C07268=1101.873,173.117,-65.868,177.861,15.228,151.662
C07269=1101.878,173.366,-65.890,177.865,15.228,151.661
C07270=1101.885,173.615,-65.912,177.869,15.227,151.660
C07271=1101.890,173.864,-65.934,177.872,15.226,151.659
C07272=1101.895,174.113,-65.957,177.876,15.226,151.658
C07273=1101.902,174.362,-65.979,177.880,15.225,151.657
C07274=1101.907,174.611,-66.002,177.883,15.224,151.656
C07275=1101.913,174.860,-66.024,177.887,15.224,151.655
C07276=1101.918,175.108,-66.046,177.890,15.223,151.654
C07277=1101.924,175.358,-66.068,177.895,15.222,151.653
C07278=1101.930,175.606,-66.091,177.898,15.222,151.652
C07279=1101.936,175.879,-66.115,177.902,15.222,151.652
C07280=1101.942,176.151,-66.140,177.906,15.221,151.650
C07281=1101.948,176.424,-66.164,177.910,15.220,151.649
C07282=1101.955,176.697,-66.188,177.914,15.219,151.648
C07283=1101.960,176.946,-66.211,177.918,15.219,151.647
C07284=1101.966,177.194,-66.234,177.922,15.218,151.647
C07285=1101.972,177.443,-66.256,177.925,15.217,151.646
C07286=1101.977,177.692,-66.279,177.929,15.217,151.645
C07287=1101.983,177.941,-66.302,177.932,15.216,151.644
C07288=1101.989,178.190,-66.323,177.936,15.215,151.643
C07289=1101.995,178.439,-66.346,177.940,15.215,151.642
C07290=1102.000,178.688,-66.369,177.943,15.214,151.641
C07291=1102.006,178.937,-66.391,177.947,15.213,151.640
C07292=1102.011,179.186,-66.414,177.952,15.213,151.639
C07293=1102.018,179.435,-66.436,177.955,15.212,151.638
C07294=1102.023,179.684,-66.458,177.959,15.211,151.637
C07295=1102.029,179.933,-66.481,177.963,15.211,151.636
C07296=1102.035,180.182,-66.504,177.966,15.210,151.635
C07297=1102.041,180.430,-66.527,177.970,15.209,151.634
C07298=1102.047,180.679,-66.550,177.973,15.208,151.633
C07299=1102.052,180.928,-66.572,177.977,15.208,151.632
C07300=1102.057,181.177,-66.594,177.981,15.207,151.631
C07301=1102.063,181.426,-66.617,177.984,15.206,151.630
C07302=1102.069,181.675,-66.640,177.989,15.205,151.629
C07303=1102.075,181.923,-66.663,177.992,15.205,151.629
C07304=1102.081,182.173,-66.685,177.996,15.204,151.628
C07305=1102.087,182.422,-66.708,178.000,15.203,151.627
C07306=1102.092,182.671,-66.731,178.004,15.203,151.626
C07307=1102.098,182.920,-66.754,178.007,15.202,151.625
C07308=1102.104,183.169,-66.777,178.011,15.201,151.624
C07309=1102.110,183.417,-66.799,178.014,15.200,151.623
C07310=1102.116,183.666,-66.822,178.018,15.200,151.622
C07311=1102.122,183.915,-66.845,178.022,15.199,151.621
C07312=1102.127,184.164,-66.868,178.026,15.198,151.620
C07313=1102.133,184.413,-66.891,178.030,15.197,151.619
C07314=1102.139,184.662,-66.914,178.034,15.197,151.618
C07315=1102.144,184.911,-66.936,178.037,15.196,151.617
C07316=1102.150,185.160,-66.959,178.041,15.195,151.616
C07317=1102.156,185.409,-66.982,178.045,15.195,151.615
C07318=1102.161,185.658,-67.005,178.048,15.194,151.614
C07319=1102.167,185.907,-67.028,178.052,15.193,151.613
C07320=1102.172,186.155,-67.050,178.056,15.193,151.612
C07321=1102.178,186.404,-67.073,178.059,15.192,151.611
C07322=1102.183,186.653,-67.097,178.064,15.191,151.610
C07323=1102.189,186.902,-67.120,178.068,15.191,151.609
C07324=1102.195,187.150,-67.143,178.071,15.190,151.608
C07325=1102.201,187.399,-67.166,178.075,15.189,151.607
C07326=1102.206,187.648,-67.189,178.079,15.189,151.606
C07327=1102.211,187.897,-67.213,178.082,15.188,151.605
C07328=1102.217,188.146,-67.236,178.086,15.187,151.604
C07329=1102.223,188.395,-67.259,178.090,15.187,151.603
C07330=1102.228,188.644,-67.282,178.093,15.186,151.603
C07331=1102.234,188.893,-67.305,178.098,15.185,151.601
C07332=1102.239,189.142,-67.328,178.101,15.185,151.601
C07333=1102.245,189.391,-67.351,178.105,15.183,151.600
C07334=1102.251,189.639,-67.375,178.109,15.183,151.599
C07335=1102.257,189.888,-67.398,178.113,15.182,151.598
C07336=1102.262,190.137,-67.421,178.116,15.182,151.597
C07337=1102.267,190.386,-67.444,178.120,15.181,151.596
C07338=1102.273,190.635,-67.467,178.124,15.181,151.595
C07339=1102.279,190.883,-67.491,178.128,15.179,151.594
C07340=1102.284,191.133,-67.514,178.132,15.179,151.593
C07341=1102.290,191.381,-67.537,178.136,15.178,151.592
C07342=1102.296,191.630,-67.560,178.139,15.177,151.591
C07343=1102.302,191.902,-67.587,178.143,15.176,151.590
C07344=1102.308,192.174,-67.611,178.147,15.176,151.589
C07345=1102.314,192.447,-67.637,178.152,15.175,151.588
C07346=1102.321,192.719,-67.663,178.156,15.174,151.586
C07347=1102.326,192.968,-67.686,178.160,15.173,151.585
C07348=1102.332,193.216,-67.710,178.163,15.173,151.585
C07349=1102.337,193.465,-67.733,178.167,15.172,151.583
C07350=1102.342,193.714,-67.756,178.172,15.171,151.582
C07351=1102.348,193.962,-67.780,178.175,15.170,151.582
C07352=1102.354,194.211,-67.803,178.179,15.170,151.580
C07353=1102.360,194.461,-67.827,178.183,15.169,151.579
C07354=1102.366,194.710,-67.850,178.186,15.168,151.579
C07355=1102.371,194.958,-67.873,178.190,15.167,151.578
C07356=1102.377,195.207,-67.898,178.195,15.167,151.576
C07357=1102.382,195.456,-67.921,178.198,15.165,151.575
C07358=1102.388,195.704,-67.944,178.202,15.165,151.575
C07359=1102.393,195.953,-67.968,178.206,15.164,151.573
C07360=1102.400,196.203,-67.991,178.210,15.164,151.572
C07361=1102.406,196.451,-68.015,178.213,15.163,151.572
C07362=1102.411,196.700,-68.038,178.218,15.162,151.570
C07363=1102.417,196.949,-68.062,178.222,15.161,151.569
C07364=1102.422,197.198,-68.086,178.225,15.160,151.568
C07365=1102.428,197.446,-68.109,178.229,15.159,151.567
C07366=1102.435,197.695,-68.133,178.233,15.159,151.566
C07367=1102.440,197.944,-68.157,178.237,15.158,151.565
C07368=1102.446,198.193,-68.180,178.241,15.157,151.564
C07369=1102.451,198.442,-68.204,178.245,15.156,151.563
C07370=1102.457,198.690,-68.228,178.248,15.155,151.562
C07371=1102.462,198.940,-68.252,178.252,15.155,151.561
C07372=1102.468,199.188,-68.275,178.257,15.154,151.560
C07373=1102.474,199.437,-68.299,178.260,15.153,151.559
C07374=1102.479,199.686,-68.322,178.264,15.152,151.558
C07375=1102.485,199.934,-68.346,178.268,15.151,151.557
C07376=1102.491,200.183,-68.371,178.272,15.150,151.556
C07377=1102.497,200.432,-68.394,178.276,15.150,151.555
C07378=1102.502,200.681,-68.418,178.280,15.149,151.554
C07379=1102.509,200.930,-68.442,178.283,15.148,151.553
C07380=1102.514,201.179,-68.465,178.288,15.147,151.552
C07381=1102.520,201.427,-68.489,178.292,15.146,151.551
C07382=1102.525,201.676,-68.513,178.295,15.145,151.550
C07383=1102.532,201.925,-68.537,178.299,15.144,151.549
C07384=1102.537,202.174,-68.561,178.304,15.144,151.548
C07385=1102.543,202.422,-68.585,178.308,15.143,151.547
C07386=1102.549,202.672,-68.609,178.311,15.142,151.546
C07387=1102.555,202.920,-68.633,178.315,15.141,151.545
C07388=1102.560,203.169,-68.657,178.319,15.141,151.544
C07389=1102.565,203.418,-68.681,178.323,15.140,151.543
C07390=1102.572,203.667,-68.705,178.327,15.139,151.542
C07391=1102.577,203.915,-68.729,178.331,15.138,151.541
C07392=1102.582,204.164,-68.753,178.334,15.137,151.540
C07393=1102.588,204.412,-68.777,178.339,15.136,151.539
C07394=1102.594,204.661,-68.801,178.343,15.136,151.538
C07395=1102.600,204.910,-68.826,178.346,15.134,151.536
C07396=1102.605,205.159,-68.849,178.350,15.134,151.535
C07397=1102.611,205.408,-68.873,178.354,15.133,151.535
C07398=1102.617,205.657,-68.898,178.359,15.133,151.533
C07399=1102.622,205.905,-68.922,178.362,15.131,151.532
C07400=1102.628,206.154,-68.945,178.366,15.131,151.531
C07401=1102.634,206.403,-68.970,178.370,15.130,151.530
C07402=1102.639,206.652,-68.994,178.374,15.129,151.529
C07403=1102.644,206.900,-69.019,178.378,15.128,151.528
C07404=1102.651,207.149,-69.043,178.382,15.127,151.527
C07405=1102.656,207.398,-69.067,178.386,15.127,151.526
C07406=1102.662,207.647,-69.092,178.390,15.125,151.525
C07407=1102.685,208.648,-69.188,178.422,15.131,151.519
C07408=1102.693,209.016,-69.225,178.428,15.131,151.518
C07409=1102.702,209.384,-69.261,178.434,15.131,151.517
C07410=1102.710,209.752,-69.297,178.439,15.131,151.516
C07411=1102.718,210.119,-69.333,178.445,15.131,151.515
C07412=1102.724,210.369,-69.358,178.448,15.132,151.514
C07413=1102.730,210.617,-69.383,178.451,15.131,151.513
C07414=1102.736,210.866,-69.408,178.455,15.131,151.512
C07415=1102.741,211.114,-69.432,178.459,15.131,151.511
C07416=1102.746,211.363,-69.456,178.462,15.131,151.511
C07417=1102.753,211.612,-69.481,178.466,15.131,151.510
C07418=1102.758,211.860,-69.506,178.470,15.131,151.509
C07419=1102.764,212.110,-69.530,178.474,15.131,151.508
C07420=1102.769,212.358,-69.555,178.477,15.131,151.507
C07421=1102.775,212.607,-69.580,178.481,15.131,151.507
C07422=1102.781,212.855,-69.604,178.485,15.132,151.506
C07423=1102.786,213.105,-69.629,178.489,15.131,151.505
C07424=1102.792,213.353,-69.654,178.493,15.132,151.504
C07425=1102.798,213.602,-69.678,178.497,15.131,151.503
C07426=1102.803,213.851,-69.703,178.500,15.132,151.503
C07427=1102.809,214.099,-69.728,178.504,15.131,151.502
C07428=1102.815,214.348,-69.752,178.508,15.132,151.501
C07429=1102.820,214.596,-69.778,178.511,15.132,151.500
C07430=1102.825,214.845,-69.802,178.515,15.132,151.499
C07431=1102.831,215.094,-69.827,178.519,15.132,151.499
C07432=1102.837,215.343,-69.852,178.522,15.132,151.498
C07433=1102.842,215.591,-69.876,178.526,15.132,151.497
C07434=1102.849,215.840,-69.902,178.530,15.132,151.496
C07435=1102.853,216.089,-69.927,178.533,15.132,151.496
C07436=1102.859,216.337,-69.952,178.537,15.132,151.495
C07437=1102.865,216.586,-69.976,178.541,15.132,151.494
C07438=1102.871,216.835,-70.001,178.544,15.132,151.493
C07439=1102.877,217.084,-70.026,178.548,15.132,151.492
C07440=1102.882,217.332,-70.051,178.552,15.132,151.492
C07441=1102.887,217.582,-70.076,178.556,15.132,151.491
C07442=1102.893,217.830,-70.101,178.559,15.132,151.490
C07443=1102.899,218.079,-70.126,178.563,15.132,151.489
C07444=1102.905,218.327,-70.151,178.567,15.132,151.488
C07445=1102.910,218.576,-70.177,178.571,15.132,151.488
C07446=1102.916,218.825,-70.201,178.574,15.132,151.487
C07447=1102.922,219.073,-70.226,178.578,15.133,151.486
C07448=1102.927,219.322,-70.251,178.581,15.132,151.485
C07449=1102.932,219.571,-70.277,178.585,15.133,151.485
C07450=1102.938,219.819,-70.302,178.589,15.132,151.484
C07451=1102.944,220.069,-70.326,178.592,15.133,151.483
C07452=1102.950,220.317,-70.351,178.596,15.132,151.482
C07453=1102.955,220.566,-70.377,178.600,15.133,151.481
C07454=1102.961,220.814,-70.402,178.604,15.132,151.480
C07455=1102.967,221.063,-70.427,178.607,15.133,151.480
C07456=1102.973,221.311,-70.452,178.612,15.133,151.479
C07457=1102.978,221.560,-70.478,178.615,15.133,151.478
C07458=1102.984,221.809,-70.503,178.619,15.133,151.477
C07459=1102.990,222.058,-70.528,178.623,15.133,151.477
C07460=1102.998,222.429,-70.566,178.628,15.133,151.475
C07461=1103.007,222.800,-70.603,178.634,15.134,151.474
C07462=1103.015,223.171,-70.641,178.639,15.133,151.473
C07463=1103.023,223.543,-70.680,178.645,15.134,151.472
C07464=1103.029,223.792,-70.704,178.649,15.134,151.471
C07465=1103.034,224.041,-70.730,178.652,15.134,151.470
C07466=1103.040,224.289,-70.756,178.656,15.134,151.470
C07467=1103.046,224.537,-70.781,178.660,15.134,151.469
C07468=1103.051,224.786,-70.806,178.663,15.134,151.468
C07469=1103.058,225.035,-70.832,178.667,15.134,151.467
C07470=1103.062,225.283,-70.857,178.671,15.135,151.466
C07471=1103.069,225.532,-70.883,178.675,15.135,151.466
C07472=1103.074,225.781,-70.909,178.679,15.135,151.465
C07473=1103.080,226.029,-70.934,178.682,15.135,151.464
C07474=1103.085,226.278,-70.960,178.686,15.135,151.463
C07475=1103.091,226.527,-70.985,178.690,15.135,151.463
C07476=1103.097,226.776,-71.011,178.693,15.136,151.462
C07477=1103.102,227.024,-71.036,178.697,15.135,151.461
C07478=1103.108,227.272,-71.062,178.701,15.136,151.460
C07479=1103.113,227.521,-71.088,178.704,15.136,151.459
C07480=1103.120,227.770,-71.113,178.708,15.136,151.459
C07481=1103.125,228.018,-71.139,178.712,15.137,151.458
C07482=1103.131,228.267,-71.164,178.716,15.137,151.457
C07483=1103.136,228.516,-71.190,178.720,15.137,151.456
C07484=1103.142,228.765,-71.215,178.724,15.137,151.455
C07485=1103.148,229.014,-71.241,178.727,15.137,151.455
C07486=1103.153,229.262,-71.267,178.731,15.137,151.454
C07487=1103.159,229.511,-71.292,178.735,15.137,151.453
C07488=1103.165,229.759,-71.319,178.738,15.137,151.452
C07489=1103.171,230.008,-71.344,178.742,15.137,151.452
C07490=1103.176,230.257,-71.370,178.746,15.137,151.451
C07491=1103.181,230.505,-71.396,178.749,15.138,151.450
C07492=1103.187,230.754,-71.421,178.754,15.138,151.449
C07493=1103.193,231.002,-71.448,178.757,15.138,151.449
C07494=1103.199,231.251,-71.473,178.761,15.138,151.448
C07495=1103.205,231.500,-71.499,178.765,15.138,151.447
C07496=1103.210,231.748,-71.524,178.768,15.139,151.446
C07497=1103.215,231.997,-71.550,178.772,15.139,151.446
C07498=1103.221,232.245,-71.577,178.776,15.139,151.445
C07499=1103.227,232.494,-71.602,178.779,15.139,151.444
C07500=1103.233,232.743,-71.628,178.783,15.140,151.443
C07501=1103.238,232.991,-71.655,178.787,15.140,151.442
C07502=1103.243,233.240,-71.680,178.791,15.140,151.442
C07503=1103.249,233.489,-71.706,178.794,15.140,151.441
C07504=1103.255,233.737,-71.732,178.798,15.140,151.440
C07505=1103.261,233.986,-71.758,178.802,15.140,151.439
C07506=1103.266,234.235,-71.784,178.805,15.141,151.439
C07507=1103.272,234.483,-71.811,178.809,15.140,151.438
C07508=1103.277,234.732,-71.837,178.813,15.141,151.437
C07509=1103.284,234.981,-71.862,178.817,15.142,151.436
C07510=1103.289,235.228,-71.888,178.821,15.142,151.436
C07511=1103.294,235.477,-71.914,178.824,15.142,151.435
C07512=1103.303,235.841,-71.953,178.830,15.142,151.434
C07513=1103.311,236.203,-71.992,178.835,15.142,151.433
C07514=1103.319,236.566,-72.030,178.841,15.143,151.432
C07515=1103.327,236.929,-72.068,178.846,15.143,151.430
C07516=1103.333,237.178,-72.094,178.850,15.144,151.430
C07517=1103.339,237.426,-72.120,178.854,15.144,151.429
C07518=1103.344,237.675,-72.146,178.858,15.144,151.428
C07519=1103.350,237.923,-72.173,178.861,15.144,151.427
C07520=1103.356,238.172,-72.199,178.865,15.144,151.427
C07521=1103.361,238.421,-72.225,178.868,15.145,151.426
C07522=1103.367,238.669,-72.252,178.873,15.145,151.425
C07523=1103.372,238.918,-72.278,178.876,15.145,151.424
C07524=1103.378,239.166,-72.305,178.880,15.146,151.424
C07525=1103.384,239.415,-72.331,178.884,15.145,151.423
C07526=1103.389,239.664,-72.357,178.887,15.146,151.422
C07527=1103.395,239.912,-72.384,178.891,15.146,151.421
C07528=1103.401,240.160,-72.410,178.895,15.147,151.421
C07529=1103.406,240.409,-72.436,178.899,15.147,151.420
C07530=1103.412,240.658,-72.463,178.903,15.147,151.419
C07531=1103.418,240.906,-72.490,178.906,15.147,151.418
C07532=1103.423,241.155,-72.516,178.910,15.147,151.418
C07533=1103.429,241.403,-72.542,178.914,15.147,151.417
C07534=1103.435,241.652,-72.569,178.918,15.148,151.416
C07535=1103.441,241.900,-72.596,178.921,15.149,151.415
C07536=1103.446,242.148,-72.622,178.925,15.149,151.415
C07537=1103.452,242.397,-72.648,178.929,15.149,151.414
C07538=1103.458,242.646,-72.675,178.932,15.149,151.413
C07539=1103.463,242.894,-72.701,178.936,15.149,151.412
C07540=1103.469,243.143,-72.728,178.940,15.150,151.412
C07541=1103.475,243.391,-72.755,178.944,15.150,151.411
C07542=1103.480,243.640,-72.781,178.947,15.150,151.410
C07543=1103.486,243.889,-72.808,178.951,15.151,151.409
C07544=1103.491,244.137,-72.835,178.955,15.151,151.409
C07545=1103.497,244.385,-72.861,178.959,15.152,151.408
C07546=1103.503,244.634,-72.888,178.963,15.152,151.407
C07547=1103.508,244.883,-72.915,178.966,15.152,151.406
C07548=1103.514,245.131,-72.942,178.970,15.152,151.406
C07549=1103.520,245.380,-72.969,178.973,15.153,151.405
C07550=1103.526,245.628,-72.995,178.978,15.154,151.404
C07551=1103.532,245.876,-73.022,178.981,15.153,151.403
C07552=1103.537,246.125,-73.049,178.985,15.154,151.403
C07553=1103.542,246.373,-73.076,178.989,15.154,151.402
C07554=1103.548,246.622,-73.103,178.992,15.154,151.401
C07555=1103.553,246.871,-73.130,178.996,15.155,151.401
C07556=1103.559,247.119,-73.156,179.000,15.155,151.400
C07557=1103.565,247.367,-73.183,179.004,15.155,151.399
C07558=1103.571,247.616,-73.210,179.007,15.156,151.398
C07559=1103.576,247.865,-73.237,179.012,15.157,151.398
C07560=1103.582,248.113,-73.264,179.015,15.157,151.397
C07561=1103.587,248.362,-73.291,179.019,15.157,151.396
C07562=1103.593,248.610,-73.318,179.022,15.157,151.396
C07563=1103.599,248.859,-73.345,179.026,15.158,151.395
C07564=1103.607,249.215,-73.384,179.031,15.158,151.394
C07565=1103.614,249.572,-73.422,179.037,15.159,151.393
C07566=1103.623,249.928,-73.461,179.042,15.160,151.392
C07567=1103.630,250.283,-73.500,179.047,15.161,151.391
C07568=1103.636,250.532,-73.527,179.051,15.161,151.390
C07569=1103.641,250.780,-73.554,179.055,15.162,151.389
C07570=1103.648,251.029,-73.582,179.059,15.162,151.389
C07571=1103.653,251.278,-73.609,179.062,15.162,151.388
C07572=1103.658,251.526,-73.636,179.066,15.162,151.387
C07573=1103.663,251.775,-73.663,179.070,15.163,151.386
C07574=1103.670,252.022,-73.690,179.074,15.163,151.386
C07575=1103.675,252.271,-73.717,179.077,15.164,151.385
C07576=1103.681,252.520,-73.744,179.081,15.164,151.384
C07577=1103.686,252.768,-73.772,179.085,15.165,151.384
C07578=1103.692,253.016,-73.799,179.089,15.165,151.383
C07579=1103.697,253.265,-73.826,179.092,15.166,151.382
C07580=1103.704,253.514,-73.854,179.096,15.166,151.382
C07581=1103.709,253.762,-73.881,179.100,15.167,151.381
C07582=1103.715,254.011,-73.908,179.104,15.167,151.380
C07583=1103.720,254.259,-73.936,179.107,15.167,151.380
C07584=1103.726,254.507,-73.963,179.111,15.168,151.379
C07585=1103.732,254.756,-73.991,179.115,15.169,151.378
C07586=1103.737,255.004,-74.018,179.119,15.169,151.377
C07587=1103.743,255.252,-74.045,179.122,15.169,151.377
C07588=1103.748,255.502,-74.073,179.126,15.170,151.376
C07589=1103.754,255.750,-74.100,179.130,15.171,151.375
C07590=1103.760,255.998,-74.128,179.133,15.171,151.375
C07591=1103.765,256.246,-74.154,179.137,15.171,151.374
C07592=1103.771,256.495,-74.183,179.141,15.172,151.373
C07593=1103.777,256.743,-74.211,179.145,15.172,151.373
C07594=1103.782,256.992,-74.237,179.149,15.172,151.372
C07595=1103.788,257.240,-74.266,179.152,15.173,151.371
C07596=1103.793,257.489,-74.293,179.156,15.174,151.370
C07597=1103.799,257.737,-74.320,179.160,15.174,151.370
C07598=1103.805,257.986,-74.348,179.164,15.174,151.369
C07599=1103.811,258.234,-74.375,179.167,15.174,151.368
C07600=1103.816,258.482,-74.403,179.171,15.175,151.367
C07601=1103.822,258.731,-74.431,179.175,15.176,151.367
C07602=1103.828,258.979,-74.458,179.178,15.176,151.366
C07603=1103.834,259.227,-74.486,179.183,15.177,151.365
C07604=1103.839,259.476,-74.514,179.186,15.177,151.365
C07605=1103.845,259.724,-74.541,179.190,15.178,151.364
C07606=1103.851,259.973,-74.569,179.193,15.178,151.363
C07607=1103.856,260.222,-74.597,179.198,15.179,151.363
C07608=1103.862,260.469,-74.624,179.201,15.179,151.362
C07609=1103.868,260.718,-74.652,179.205,15.179,151.361
C07610=1103.874,260.966,-74.680,179.209,15.180,151.361
C07611=1103.879,261.215,-74.708,179.212,15.181,151.360
C07612=1103.885,261.463,-74.735,179.216,15.181,151.359
C07613=1103.891,261.711,-74.763,179.220,15.182,151.358
C07614=1103.897,261.960,-74.792,179.224,15.182,151.358
C07615=1103.903,262.208,-74.819,179.227,15.183,151.357
C07616=1103.910,262.561,-74.859,179.233,15.183,151.356
C07617=1103.918,262.915,-74.898,179.238,15.185,151.355
C07618=1103.927,263.268,-74.938,179.243,15.185,151.354
C07619=1103.935,263.622,-74.977,179.249,15.186,151.353
C07620=1103.941,263.871,-75.006,179.252,15.186,151.352
C07621=1103.946,264.119,-75.034,179.257,15.187,151.352
C07622=1103.953,264.367,-75.061,179.260,15.187,151.351
C07623=1103.958,264.615,-75.089,179.264,15.187,151.350
C07624=1103.964,264.864,-75.118,179.268,15.189,151.350
C07625=1103.970,265.112,-75.146,179.271,15.189,151.349
C07626=1103.975,265.361,-75.174,179.275,15.190,151.348
C07627=1103.981,265.609,-75.202,179.279,15.191,151.348
C07628=1103.986,265.857,-75.230,179.283,15.191,151.347
C07629=1103.992,266.106,-75.258,179.286,15.191,151.346
C07630=1103.997,266.354,-75.286,179.290,15.193,151.346
C07631=1104.003,266.602,-75.315,179.294,15.193,151.345
C07632=1104.009,266.850,-75.343,179.297,15.193,151.344
C07633=1104.015,267.099,-75.371,179.301,15.194,151.344
C07634=1104.020,267.347,-75.400,179.305,15.194,151.343
C07635=1104.026,267.595,-75.428,179.308,15.195,151.342
C07636=1104.032,267.843,-75.456,179.312,15.196,151.342
C07637=1104.038,268.092,-75.484,179.316,15.197,151.341
C07638=1104.043,268.340,-75.512,179.319,15.197,151.340
C07639=1104.049,268.589,-75.540,179.324,15.198,151.340
C07640=1104.054,268.837,-75.568,179.327,15.198,151.339
C07641=1104.060,269.085,-75.597,179.330,15.199,151.339
C07642=1104.066,269.334,-75.626,179.335,15.200,151.338
C07643=1104.072,269.582,-75.654,179.338,15.200,151.337
C07644=1104.078,269.831,-75.682,179.342,15.201,151.336
C07645=1104.083,270.079,-75.710,179.346,15.202,151.336
C07646=1104.088,270.327,-75.740,179.349,15.202,151.335
C07647=1104.094,270.575,-75.768,179.353,15.203,151.335
C07648=1104.100,270.824,-75.796,179.357,15.204,151.334
C07649=1104.105,271.071,-75.825,179.360,15.204,151.333
C07650=1104.111,271.320,-75.853,179.364,15.205,151.333
C07651=1104.117,271.569,-75.881,179.368,15.206,151.332
C07652=1104.122,271.817,-75.910,179.372,15.206,151.331
C07653=1104.128,272.065,-75.939,179.375,15.207,151.331
C07654=1104.134,272.313,-75.967,179.379,15.208,151.330
C07655=1104.140,272.562,-75.996,179.383,15.208,151.329
C07656=1104.145,272.810,-76.024,179.386,15.209,151.329
C07657=1104.151,273.058,-76.052,179.390,15.210,151.328
C07658=1104.157,273.307,-76.082,179.394,15.211,151.327
C07659=1104.162,273.555,-76.110,179.397,15.211,151.327
C07660=1104.168,273.803,-76.139,179.401,15.212,151.326
C07661=1104.174,274.052,-76.167,179.405,15.213,151.326
C07662=1104.179,274.300,-76.196,179.409,15.213,151.325
C07663=1104.185,274.548,-76.225,179.413,15.215,151.324
C07664=1104.191,274.796,-76.253,179.416,15.215,151.324
C07665=1104.196,275.045,-76.282,179.419,15.216,151.323
C07666=1104.202,275.293,-76.311,179.424,15.217,151.322
C07667=1104.207,275.541,-76.339,179.427,15.217,151.322
C07668=1104.216,275.897,-76.381,179.433,15.218,151.321
C07669=1104.224,276.253,-76.422,179.438,15.219,151.320
C07670=1104.232,276.610,-76.463,179.443,15.221,151.319
C07671=1104.240,276.966,-76.505,179.449,15.222,151.318
C07672=1104.245,277.214,-76.534,179.452,15.222,151.318
C07673=1104.252,277.462,-76.563,179.456,15.224,151.317
C07674=1104.257,277.711,-76.592,179.460,15.224,151.316
C07675=1104.262,277.959,-76.620,179.463,15.224,151.316
C07676=1104.269,278.207,-76.650,179.467,15.226,151.315
C07677=1104.274,278.456,-76.678,179.471,15.226,151.315
C07678=1104.280,278.703,-76.707,179.475,15.228,151.314
C07679=1104.285,278.952,-76.737,179.478,15.228,151.313
C07680=1104.291,279.200,-76.766,179.482,15.229,151.313
C07681=1104.296,279.448,-76.794,179.486,15.230,151.312
C07682=1104.302,279.696,-76.823,179.489,15.230,151.312
C07683=1104.308,279.945,-76.853,179.493,15.231,151.311
C07684=1104.314,280.193,-76.882,179.496,15.232,151.310
C07685=1104.319,280.441,-76.910,179.500,15.233,151.310
C07686=1104.325,280.690,-76.940,179.504,15.233,151.309
C07687=1104.331,280.938,-76.969,179.508,15.235,151.309
C07688=1104.337,281.186,-76.998,179.511,15.235,151.308
C07689=1104.342,281.434,-77.027,179.515,15.236,151.307
C07690=1104.348,281.682,-77.057,179.519,15.237,151.307
C07691=1104.353,281.930,-77.086,179.522,15.238,151.306
C07692=1104.359,282.179,-77.115,179.526,15.239,151.306
C07693=1104.364,282.427,-77.144,179.530,15.240,151.305
C07694=1104.370,282.675,-77.173,179.534,15.241,151.304
C07695=1104.376,282.923,-77.203,179.537,15.242,151.304
C07696=1104.381,283.172,-77.232,179.541,15.243,151.303
C07697=1104.387,283.419,-77.261,179.544,15.243,151.303
C07698=1104.392,283.668,-77.290,179.548,15.244,151.302
C07699=1104.398,283.916,-77.320,179.552,15.245,151.302
C07700=1104.404,284.164,-77.349,179.555,15.246,151.301
C07701=1104.410,284.413,-77.379,179.559,15.247,151.300
C07702=1104.415,284.661,-77.408,179.562,15.248,151.300
C07703=1104.421,284.909,-77.437,179.567,15.249,151.299
C07704=1104.426,285.157,-77.467,179.570,15.250,151.299
C07705=1104.432,285.406,-77.496,179.574,15.251,151.298
C07706=1104.438,285.654,-77.525,179.577,15.251,151.297
C07707=1104.444,285.902,-77.555,179.581,15.253,151.297
C07708=1104.449,286.149,-77.585,179.584,15.254,151.296
C07709=1104.455,286.397,-77.614,179.589,15.255,151.296
C07710=1104.461,286.646,-77.644,179.592,15.255,151.295
C07711=1104.466,286.894,-77.673,179.596,15.257,151.295
C07712=1104.472,287.143,-77.703,179.599,15.257,151.294
C07713=1104.478,287.391,-77.732,179.603,15.258,151.294
C07714=1104.484,287.639,-77.762,179.606,15.259,151.293
C07715=1104.489,287.886,-77.792,179.611,15.260,151.292
C07716=1104.494,288.135,-77.821,179.614,15.261,151.292
C07717=1104.500,288.383,-77.850,179.618,15.262,151.291
C07718=1104.506,288.631,-77.881,179.621,15.263,151.291
C07719=1104.512,288.879,-77.910,179.625,15.264,151.290
C07720=1104.520,289.245,-77.953,179.631,15.266,151.289
C07721=1104.529,289.611,-77.998,179.636,15.267,151.288
C07722=1104.537,289.976,-78.041,179.641,15.268,151.288
C07723=1104.545,290.341,-78.085,179.646,15.270,151.287
C07724=1104.551,290.590,-78.115,179.650,15.271,151.286
C07725=1104.557,290.838,-78.145,179.653,15.272,151.286
C07726=1104.562,291.086,-78.175,179.658,15.273,151.285
C07727=1104.568,291.335,-78.205,179.661,15.274,151.285
C07728=1104.574,291.582,-78.234,179.665,15.275,151.284
C07729=1104.580,291.831,-78.264,179.668,15.276,151.284
C07730=1104.586,292.078,-78.294,179.672,15.277,151.283
C07731=1104.591,292.327,-78.324,179.676,15.279,151.283
C07732=1104.597,292.575,-78.354,179.679,15.279,151.282
C07733=1104.602,292.823,-78.384,179.683,15.281,151.281
C07734=1104.608,293.072,-78.414,179.687,15.281,151.281
C07735=1104.614,293.319,-78.444,179.690,15.283,151.280
C07736=1104.619,293.568,-78.474,179.694,15.284,151.280
C07737=1104.625,293.816,-78.504,179.698,15.285,151.279
C07738=1104.631,294.063,-78.534,179.701,15.286,151.279
C07739=1104.636,294.312,-78.564,179.705,15.287,151.278
C07740=1104.642,294.560,-78.594,179.708,15.288,151.278
C07741=1104.648,294.808,-78.624,179.712,15.289,151.277
C07742=1104.654,295.056,-78.654,179.715,15.290,151.277
C07743=1104.659,295.304,-78.685,179.719,15.291,151.276
C07744=1104.665,295.552,-78.714,179.723,15.293,151.276
C07745=1104.671,295.800,-78.745,179.726,15.294,151.275
C07746=1104.676,296.048,-78.774,179.730,15.295,151.275
C07747=1104.682,296.296,-78.805,179.734,15.296,151.274
C07748=1104.688,296.544,-78.835,179.738,15.297,151.274
C07749=1104.693,296.792,-78.866,179.741,15.298,151.273
C07750=1104.698,297.041,-78.895,179.745,15.299,151.273
C07751=1104.704,297.289,-78.926,179.749,15.301,151.272
C07752=1104.710,297.536,-78.956,179.752,15.302,151.272
C07753=1104.716,297.785,-78.986,179.756,15.303,151.271
C07754=1104.721,298.033,-79.016,179.759,15.304,151.271
C07755=1104.727,298.280,-79.047,179.763,15.305,151.270
C07756=1104.732,298.529,-79.077,179.767,15.307,151.270
C07757=1104.738,298.776,-79.108,179.770,15.308,151.269
C07758=1104.744,299.025,-79.137,179.774,15.309,151.269
C07759=1104.749,299.273,-79.168,179.777,15.310,151.268
C07760=1104.754,299.521,-79.199,179.781,15.312,151.268
C07761=1104.760,299.769,-79.229,179.785,15.313,151.267
C07762=1104.766,300.016,-79.259,179.788,15.314,151.267
C07763=1104.771,300.265,-79.290,179.791,15.316,151.266
C07764=1104.777,300.512,-79.321,179.795,15.316,151.266
C07765=1104.783,300.761,-79.350,179.799,15.318,151.265
C07766=1104.788,301.009,-79.381,179.803,15.319,151.265
C07767=1104.794,301.257,-79.412,179.805,15.321,151.265
C07768=1104.799,301.506,-79.443,179.809,15.322,151.264
C07769=1104.805,301.753,-79.473,179.813,15.323,151.264
C07770=1104.811,302.001,-79.504,179.816,15.324,151.263
C07771=1104.816,302.249,-79.535,179.820,15.326,151.263
C07772=1104.824,302.628,-79.581,179.825,15.327,151.262
C07773=1104.834,303.008,-79.628,179.831,15.330,151.261
C07774=1104.841,303.388,-79.675,179.837,15.332,151.261
C07775=1104.851,303.767,-79.723,179.842,15.334,151.260
C07776=1104.856,304.015,-79.753,179.846,15.335,151.259
C07777=1104.862,304.263,-79.784,179.849,15.336,151.259
C07778=1104.868,304.511,-79.814,179.853,15.338,151.259
C07779=1104.873,304.759,-79.845,179.857,15.339,151.258
C07780=1104.879,305.007,-79.876,179.859,15.341,151.258
C07781=1104.884,305.255,-79.907,179.863,15.342,151.257
C07782=1104.890,305.503,-79.938,179.867,15.343,151.257
C07783=1104.895,305.751,-79.969,179.870,15.345,151.256
C07784=1104.901,305.999,-79.999,179.874,15.346,151.256
C07785=1104.907,306.247,-80.030,179.878,15.348,151.255
C07786=1104.913,306.495,-80.061,179.881,15.349,151.255
C07787=1104.918,306.743,-80.092,179.885,15.350,151.255
C07788=1104.924,306.991,-80.123,179.889,15.352,151.254
C07789=1104.929,307.239,-80.154,179.892,15.353,151.254
C07790=1104.936,307.487,-80.185,179.896,15.354,151.253
C07791=1104.941,307.735,-80.216,179.899,15.356,151.253
C07792=1104.947,307.983,-80.246,179.902,15.357,151.252
C07793=1104.952,308.230,-80.278,179.906,15.358,151.252
C07794=1104.958,308.479,-80.309,179.910,15.360,151.252
C07795=1104.963,308.727,-80.340,179.913,15.361,151.251
C07796=1104.970,308.974,-80.371,179.917,15.363,151.251
C07797=1104.975,309.223,-80.402,179.921,15.364,151.250
C07798=1104.981,309.471,-80.433,179.924,15.366,151.250
C07799=1104.986,309.718,-80.464,179.927,15.367,151.249
C07800=1104.992,309.967,-80.496,179.931,15.369,151.249
C07801=1104.998,310.214,-80.527,179.935,15.370,151.249
C07802=1105.003,310.462,-80.558,179.938,15.371,151.248
C07803=1105.010,310.710,-80.589,179.942,15.373,151.248
C07804=1105.015,310.958,-80.620,179.946,15.375,151.247
C07805=1105.021,311.206,-80.652,179.949,15.376,151.247
C07806=1105.027,311.454,-80.682,179.953,15.377,151.246
C07807=1105.032,311.702,-80.714,179.956,15.379,151.246
C07808=1105.038,311.950,-80.744,179.959,15.380,151.246
C07809=1105.044,312.198,-80.776,179.963,15.382,151.245
C07810=1105.049,312.446,-80.807,179.967,15.383,151.245
C07811=1105.056,312.694,-80.839,179.970,15.384,151.244
C07812=1105.061,312.942,-80.870,179.973,15.386,151.244
C07813=1105.067,313.190,-80.902,179.977,15.388,151.244
C07814=1105.073,313.437,-80.933,179.981,15.390,151.243
C07815=1105.078,313.686,-80.964,179.984,15.390,151.243
C07816=1105.084,313.934,-80.996,179.988,15.392,151.242
C07817=1105.090,314.181,-81.027,179.992,15.394,151.242
C07818=1105.096,314.430,-81.058,179.994,15.395,151.242
C07819=1105.101,314.677,-81.090,179.998,15.397,151.241
C07820=1105.107,314.926,-81.122,-179.998,15.398,151.241
C07821=1105.113,315.173,-81.152,-179.994,15.400,151.240
C07822=1105.119,315.422,-81.184,-179.992,15.401,151.240
C07823=1105.125,315.669,-81.216,-179.988,15.403,151.240
C07824=1105.133,316.051,-81.265,-179.982,15.406,151.239
C07825=1105.141,316.434,-81.313,-179.977,15.408,151.239
C07826=1105.150,316.816,-81.362,-179.972,15.411,151.238
C07827=1105.159,317.198,-81.411,-179.967,15.413,151.238
C07828=1105.164,317.445,-81.442,-179.963,15.415,151.237
C07829=1105.170,317.693,-81.474,-179.959,15.417,151.237
C07830=1105.176,317.941,-81.505,-179.956,15.419,151.236
C07831=1105.181,318.189,-81.537,-179.953,15.420,151.236
C07832=1105.187,318.437,-81.569,-179.949,15.422,151.236
C07833=1105.192,318.685,-81.601,-179.945,15.423,151.236
C07834=1105.198,318.933,-81.633,-179.942,15.425,151.235
C07835=1105.204,319.180,-81.664,-179.939,15.427,151.235
C07836=1105.209,319.429,-81.697,-179.935,15.428,151.235
C07837=1105.214,319.676,-81.729,-179.932,15.430,151.234
C07838=1105.220,319.925,-81.761,-179.928,15.432,151.234
C07839=1105.226,320.172,-81.792,-179.925,15.434,151.234
C07840=1105.232,320.420,-81.824,-179.922,15.435,151.233
C07841=1105.237,320.668,-81.856,-179.918,15.437,151.233
C07842=1105.243,320.916,-81.888,-179.915,15.439,151.233
C07843=1105.248,321.164,-81.920,-179.911,15.441,151.232
C07844=1105.254,321.412,-81.952,-179.908,15.443,151.232
C07845=1105.260,321.659,-81.983,-179.905,15.444,151.232
C07846=1105.266,321.908,-82.015,-179.901,15.446,151.231
C07847=1105.270,322.155,-82.048,-179.897,15.448,151.231
C07848=1105.276,322.404,-82.080,-179.894,15.450,151.231
C07849=1105.282,322.652,-82.112,-179.890,15.452,151.230
C07850=1105.288,322.899,-82.143,-179.887,15.453,151.230
C07851=1105.294,323.148,-82.175,-179.884,15.455,151.230
C07852=1105.299,323.394,-82.208,-179.880,15.457,151.230
C07853=1105.305,323.643,-82.240,-179.877,15.459,151.229
C07854=1105.310,323.890,-82.272,-179.873,15.461,151.229
C07855=1105.316,324.139,-82.304,-179.870,15.463,151.229
C07856=1105.322,324.387,-82.336,-179.867,15.464,151.228
C07857=1105.328,324.634,-82.369,-179.863,15.466,151.228
C07858=1105.333,324.882,-82.401,-179.860,15.468,151.228
C07859=1105.339,325.131,-82.433,-179.856,15.470,151.228
C07860=1105.344,325.378,-82.465,-179.853,15.472,151.227
C07861=1105.351,325.626,-82.498,-179.849,15.474,151.227
C07862=1105.357,325.874,-82.530,-179.847,15.475,151.227
C07863=1105.361,326.122,-82.562,-179.843,15.477,151.226
C07864=1105.368,326.369,-82.595,-179.839,15.479,151.226
C07865=1105.374,326.617,-82.627,-179.836,15.481,151.226
C07866=1105.379,326.865,-82.658,-179.832,15.483,151.226
C07867=1105.385,327.113,-82.692,-179.829,15.485,151.225
C07868=1105.391,327.361,-82.724,-179.825,15.487,151.225
C07869=1105.396,327.609,-82.755,-179.823,15.489,151.225
C07870=1105.402,327.856,-82.788,-179.819,15.491,151.225
C07871=1105.407,328.105,-82.821,-179.815,15.493,151.224
C07872=1105.414,328.352,-82.853,-179.812,15.495,151.224
C07873=1105.419,328.600,-82.885,-179.809,15.497,151.224
C07874=1105.425,328.848,-82.918,-179.805,15.499,151.223
C07875=1105.431,329.096,-82.950,-179.802,15.501,151.223
C07876=1105.440,329.470,-83.000,-179.796,15.504,151.223
C07877=1105.448,329.846,-83.048,-179.792,15.506,151.222
C07878=1105.456,330.221,-83.098,-179.787,15.509,151.222
C07879=1105.465,330.596,-83.147,-179.781,15.512,151.222
C07880=1105.471,330.843,-83.180,-179.778,15.514,151.221
C07881=1105.477,331.091,-83.213,-179.775,15.516,151.221
C07882=1105.483,331.339,-83.245,-179.771,15.518,151.221
C07883=1105.489,331.587,-83.278,-179.768,15.521,151.221
C07884=1105.494,331.836,-83.310,-179.764,15.522,151.220
C07885=1105.500,332.082,-83.343,-179.761,15.525,151.220
C07886=1105.506,332.330,-83.376,-179.757,15.527,151.220
C07887=1105.512,332.579,-83.408,-179.755,15.528,151.220
C07888=1105.517,332.826,-83.441,-179.751,15.531,151.220
C07889=1105.523,333.074,-83.474,-179.748,15.532,151.219
C07890=1105.528,333.321,-83.507,-179.744,15.535,151.219
C07891=1105.534,333.570,-83.540,-179.741,15.537,151.219
C07892=1105.540,333.817,-83.572,-179.738,15.539,151.219
C07893=1105.545,334.065,-83.606,-179.734,15.541,151.219
C07894=1105.551,334.312,-83.638,-179.731,15.543,151.218
C07895=1105.556,334.561,-83.671,-179.728,15.546,151.218
C07896=1105.562,334.809,-83.704,-179.724,15.548,151.218
C07897=1105.568,335.056,-83.737,-179.721,15.550,151.218
C07898=1105.574,335.304,-83.770,-179.717,15.552,151.218
C07899=1105.579,335.552,-83.804,-179.714,15.554,151.218
C07900=1105.585,335.799,-83.835,-179.711,15.557,151.217
C07901=1105.590,336.047,-83.869,-179.708,15.559,151.217
C07902=1105.597,336.295,-83.901,-179.704,15.561,151.217
C07903=1105.602,336.543,-83.935,-179.701,15.563,151.217
C07904=1105.608,336.791,-83.968,-179.697,15.565,151.217
C07905=1105.614,337.038,-84.001,-179.694,15.568,151.216
C07906=1105.620,337.286,-84.034,-179.691,15.570,151.216
C07907=1105.625,337.534,-84.067,-179.688,15.572,151.216
C07908=1105.630,337.781,-84.100,-179.684,15.575,151.216
C07909=1105.636,338.029,-84.133,-179.681,15.577,151.216
C07910=1105.642,338.277,-84.166,-179.678,15.579,151.216
C07911=1105.647,338.525,-84.200,-179.674,15.581,151.216
C07912=1105.654,338.772,-84.233,-179.671,15.584,151.215
C07913=1105.659,339.020,-84.266,-179.668,15.586,151.215
C07914=1105.665,339.268,-84.299,-179.665,15.588,151.215
C07915=1105.670,339.516,-84.333,-179.661,15.591,151.215
C07916=1105.676,339.764,-84.366,-179.658,15.593,151.215
C07917=1105.682,340.012,-84.399,-179.655,15.595,151.215
C07918=1105.687,340.259,-84.432,-179.651,15.597,151.215
C07919=1105.693,340.507,-84.465,-179.648,15.600,151.215
C07920=1105.699,340.754,-84.499,-179.645,15.602,151.214
C07921=1105.704,341.002,-84.532,-179.642,15.605,151.214
C07922=1105.710,341.250,-84.566,-179.639,15.607,151.214
C07923=1105.715,341.498,-84.599,-179.635,15.609,151.214
C07924=1105.721,341.746,-84.632,-179.632,15.613,151.214
C07925=1105.727,341.993,-84.666,-179.628,15.615,151.214
C07926=1105.732,342.241,-84.700,-179.625,15.617,151.214
C07927=1105.739,342.488,-84.732,-179.622,15.620,151.214
C07928=1105.747,342.857,-84.783,-179.617,15.623,151.213
C07929=1105.756,343.226,-84.833,-179.612,15.627,151.213
C07930=1105.764,343.595,-84.883,-179.607,15.630,151.213
C07931=1105.772,343.964,-84.932,-179.603,15.634,151.213
C07932=1105.778,344.212,-84.966,-179.600,15.637,151.213
C07933=1105.784,344.460,-85.000,-179.596,15.639,151.213
C07934=1105.789,344.707,-85.034,-179.593,15.641,151.213
C07935=1105.795,344.955,-85.067,-179.590,15.644,151.213
C07936=1105.801,345.203,-85.100,-179.586,15.647,151.213
C07937=1105.806,345.450,-85.134,-179.583,15.650,151.213
C07938=1105.812,345.698,-85.168,-179.580,15.652,151.213
C07939=1105.818,345.945,-85.202,-179.577,15.655,151.213
C07940=1105.823,346.193,-85.235,-179.574,15.657,151.212
C07941=1105.829,346.440,-85.269,-179.571,15.660,151.212
C07942=1105.835,346.688,-85.302,-179.567,15.662,151.212
C07943=1105.841,346.936,-85.337,-179.564,15.665,151.212
C07944=1105.846,347.184,-85.370,-179.560,15.667,151.212
C07945=1105.851,347.431,-85.405,-179.557,15.670,151.212
C07946=1105.857,347.679,-85.438,-179.554,15.673,151.212
C07947=1105.863,347.926,-85.472,-179.551,15.675,151.212
C07948=1105.868,348.174,-85.505,-179.548,15.678,151.212
C07949=1105.874,348.421,-85.539,-179.545,15.680,151.212
C07950=1105.880,348.669,-85.573,-179.542,15.683,151.212
C07951=1105.885,348.918,-85.608,-179.538,15.686,151.212
C07952=1105.891,349.165,-85.642,-179.535,15.689,151.212
C07953=1105.897,349.413,-85.675,-179.532,15.691,151.212
C07954=1105.903,349.660,-85.709,-179.529,15.694,151.212
C07955=1105.909,349.907,-85.743,-179.526,15.696,151.212
C07956=1105.914,350.155,-85.778,-179.522,15.700,151.212
C07957=1105.919,350.403,-85.811,-179.519,15.703,151.212
C07958=1105.925,350.650,-85.845,-179.516,15.705,151.212
C07959=1105.931,350.897,-85.879,-179.513,15.708,151.212
C07960=1105.937,351.146,-85.914,-179.510,15.711,151.212
C07961=1105.942,351.394,-85.948,-179.507,15.713,151.212
C07962=1105.948,351.641,-85.982,-179.503,15.716,151.212
C07963=1105.954,351.888,-86.016,-179.500,15.719,151.212
C07964=1105.959,352.136,-86.050,-179.497,15.722,151.212
C07965=1105.965,352.383,-86.084,-179.494,15.724,151.212
C07966=1105.971,352.632,-86.118,-179.491,15.728,151.212
C07967=1105.976,352.879,-86.153,-179.488,15.730,151.212
C07968=1105.982,353.127,-86.187,-179.485,15.733,151.212
C07969=1105.988,353.374,-86.221,-179.482,15.736,151.212
C07970=1105.993,353.621,-86.256,-179.479,15.738,151.212
C07971=1105.999,353.869,-86.290,-179.475,15.742,151.212
C07972=1106.005,354.117,-86.324,-179.472,15.745,151.212
C07973=1106.011,354.364,-86.359,-179.469,15.747,151.212
C07974=1106.016,354.612,-86.393,-179.466,15.750,151.212
C07975=1106.022,354.859,-86.427,-179.463,15.753,151.212
C07976=1106.027,355.107,-86.461,-179.460,15.756,151.212
C07977=1106.033,355.355,-86.496,-179.457,15.759,151.213
C07978=1106.039,355.602,-86.530,-179.454,15.762,151.213
C07979=1106.045,355.849,-86.565,-179.450,15.765,151.213
C07980=1106.053,356.220,-86.617,-179.446,15.770,151.213
C07981=1106.061,356.592,-86.668,-179.441,15.774,151.213
C07982=1106.070,356.962,-86.719,-179.437,15.779,151.213
C07983=1106.078,357.333,-86.771,-179.432,15.783,151.213
C07984=1106.085,357.581,-86.806,-179.429,15.787,151.213
C07985=1106.090,357.829,-86.840,-179.426,15.789,151.213
C07986=1106.095,358.077,-86.875,-179.423,15.792,151.214
C07987=1106.101,358.323,-86.910,-179.420,15.796,151.214
C07988=1106.107,358.572,-86.945,-179.417,15.798,151.214
C07989=1106.113,358.819,-86.979,-179.414,15.801,151.214
C07990=1106.118,359.066,-87.014,-179.411,15.804,151.214
C07991=1106.124,359.314,-87.049,-179.408,15.808,151.214
C07992=1106.130,359.561,-87.083,-179.405,15.811,151.214
C07993=1106.135,359.809,-87.117,-179.402,15.814,151.214
C07994=1106.141,360.057,-87.152,-179.399,15.817,151.215
C07995=1106.147,360.304,-87.188,-179.396,15.820,151.215
C07996=1106.152,360.551,-87.222,-179.393,15.823,151.215
C07997=1106.158,360.799,-87.256,-179.390,15.827,151.215
C07998=1106.164,361.046,-87.292,-179.387,15.830,151.215
C07999=1106.169,361.294,-87.326,-179.384,15.833,151.215
C08000=1106.175,361.541,-87.362,-179.380,15.836,151.215
C08001=1106.181,361.789,-87.397,-179.378,15.839,151.216
C08002=1106.187,362.036,-87.431,-179.375,15.842,151.216
C08003=1106.192,362.283,-87.466,-179.371,15.846,151.216
C08004=1106.198,362.532,-87.501,-179.369,15.849,151.216
C08005=1106.204,362.778,-87.536,-179.365,15.853,151.216
C08006=1106.209,363.026,-87.570,-179.363,15.856,151.216
C08007=1106.215,363.273,-87.606,-179.360,15.859,151.217
C08008=1106.220,363.521,-87.641,-179.357,15.863,151.217
C08009=1106.226,363.768,-87.676,-179.354,15.866,151.217
C08010=1106.232,364.016,-87.711,-179.351,15.869,151.217
C08011=1106.237,364.263,-87.746,-179.348,15.872,151.217
C08012=1106.243,364.511,-87.781,-179.345,15.876,151.218
C08013=1106.249,364.758,-87.816,-179.342,15.879,151.218
C08014=1106.255,365.005,-87.851,-179.339,15.882,151.218
C08015=1106.260,365.253,-87.886,-179.336,15.885,151.218
C08016=1106.266,365.500,-87.921,-179.333,15.889,151.218
C08017=1106.272,365.749,-87.957,-179.330,15.892,151.219
C08018=1106.277,365.995,-87.992,-179.327,15.896,151.219
C08019=1106.283,366.242,-88.027,-179.324,15.899,151.219
C08020=1106.289,366.490,-88.062,-179.321,15.903,151.219
C08021=1106.294,366.737,-88.097,-179.319,15.906,151.220
C08022=1106.300,366.985,-88.133,-179.316,15.909,151.220
C08023=1106.306,367.232,-88.168,-179.312,15.913,151.220
C08024=1106.311,367.480,-88.203,-179.310,15.916,151.220
C08025=1106.317,367.727,-88.238,-179.307,15.920,151.220
C08026=1106.322,367.974,-88.274,-179.304,15.924,151.221
C08027=1106.328,368.222,-88.310,-179.301,15.927,151.221
C08028=1106.334,368.469,-88.345,-179.298,15.931,151.221
C08029=1106.339,368.717,-88.380,-179.295,15.935,151.222
C08030=1106.345,368.964,-88.415,-179.292,15.938,151.222
C08031=1106.350,369.211,-88.451,-179.289,15.942,151.222
C08032=1106.356,369.434,-88.483,-179.287,15.945,151.222
C08033=1106.361,369.657,-88.514,-179.284,15.948,151.223
C08034=1106.366,369.880,-88.547,-179.282,15.951,151.223
C08035=1106.371,370.103,-88.578,-179.279,15.955,151.223
C08036=1106.377,370.326,-88.611,-179.277,15.958,151.223
C08037=1106.381,370.549,-88.642,-179.274,15.961,151.224
C08038=1106.387,370.772,-88.675,-179.272,15.964,151.224
C08039=1106.392,370.995,-88.707,-179.269,15.968,151.224
C08040=1106.398,371.242,-88.743,-179.266,15.972,151.225
C08041=1106.403,371.489,-88.778,-179.263,15.975,151.225
C08042=1106.409,371.737,-88.814,-179.260,15.979,151.225
C08043=1106.415,371.984,-88.849,-179.258,15.982,151.225
C08044=1106.421,372.232,-88.885,-179.255,15.986,151.226
C08045=1106.425,372.479,-88.921,-179.252,15.990,151.226
C08046=1106.431,372.726,-88.957,-179.249,15.994,151.227
C08047=1106.437,372.973,-88.992,-179.246,15.997,151.227
C08048=1106.443,373.221,-89.028,-179.243,16.001,151.227
C08049=1106.448,373.468,-89.063,-179.241,16.005,151.228
C08050=1106.454,373.716,-89.099,-179.238,16.009,151.228
C08051=1106.460,373.963,-89.134,-179.235,16.012,151.228
C08052=1106.466,374.210,-89.171,-179.232,16.016,151.229
C08053=1106.472,374.457,-89.206,-179.230,16.020,151.229
C08054=1106.477,374.705,-89.242,-179.227,16.024,151.229
C08055=1106.483,374.952,-89.278,-179.224,16.028,151.230
C08056=1106.488,375.199,-89.313,-179.221,16.032,151.230
C08057=1106.494,375.447,-89.350,-179.219,16.036,151.231
C08058=1106.499,375.694,-89.386,-179.216,16.040,151.231
C08059=1106.505,375.941,-89.421,-179.213,16.044,151.231
C08060=1106.511,376.188,-89.457,-179.210,16.048,151.232
C08061=1106.516,376.436,-89.494,-179.208,16.052,151.232
C08062=1106.522,376.683,-89.529,-179.205,16.056,151.233
C08063=1106.528,376.930,-89.565,-179.202,16.059,151.233
C08064=1106.533,377.178,-89.602,-179.200,16.064,151.233
C08065=1106.539,377.425,-89.637,-179.197,16.068,151.234
C08066=1106.545,377.672,-89.674,-179.194,16.071,151.234
C08067=1106.550,377.919,-89.710,-179.191,16.076,151.235
C08068=1106.556,378.167,-89.745,-179.188,16.080,151.235
C08069=1106.562,378.414,-89.782,-179.186,16.084,151.236
C08070=1106.567,378.661,-89.818,-179.183,16.088,151.236
C08071=1106.573,378.908,-89.854,-179.180,16.092,151.237
C08072=1106.578,379.125,-89.886,-179.178,16.096,151.237
C08073=1106.583,379.342,-89.918,-179.176,16.099,151.237
C08074=1106.587,379.559,-89.950,-179.173,16.103,151.238
C08075=1106.593,379.777,-89.981,-179.171,16.107,151.238
C08076=1106.598,379.994,-90.013,-179.169,16.110,151.238
C08077=1106.603,380.211,-90.045,-179.167,16.114,151.239
C08078=1106.608,380.429,-90.077,-179.164,16.117,151.239
C08079=1106.613,380.646,-90.109,-179.162,16.121,151.240
C08080=1106.619,380.894,-90.145,-179.159,16.125,151.240
C08081=1106.624,381.140,-90.182,-179.156,16.130,151.241
C08082=1106.630,381.387,-90.218,-179.154,16.134,151.241
C08083=1106.635,381.635,-90.254,-179.151,16.138,151.242
C08084=1106.641,381.882,-90.290,-179.148,16.142,151.242
C08085=1106.648,382.129,-90.327,-179.145,16.147,151.243
C08086=1106.653,382.377,-90.363,-179.143,16.151,151.243
C08087=1106.659,382.624,-90.400,-179.141,16.155,151.244
C08088=1106.668,383.036,-90.461,-179.136,16.162,151.245
C08089=1106.678,383.449,-90.521,-179.132,16.170,151.246
C08090=1106.687,383.861,-90.582,-179.127,16.177,151.246
C08091=1106.696,384.274,-90.643,-179.123,16.185,151.248
C08092=1106.702,384.521,-90.680,-179.121,16.188,151.248
C08093=1106.707,384.768,-90.716,-179.118,16.193,151.249
C08094=1106.713,385.015,-90.753,-179.116,16.198,151.249
C08095=1106.719,385.262,-90.790,-179.113,16.202,151.250
C08096=1106.724,385.509,-90.827,-179.110,16.207,151.250
C08097=1106.729,385.757,-90.863,-179.108,16.211,151.251
C08098=1106.736,386.004,-90.899,-179.105,16.216,151.252
C08099=1106.741,386.251,-90.936,-179.103,16.220,151.252
C08100=1106.746,386.498,-90.973,-179.100,16.225,151.253
C08101=1106.753,386.745,-91.009,-179.098,16.230,151.253
C08102=1106.758,386.992,-91.047,-179.095,16.234,151.254
C08103=1106.764,387.240,-91.084,-179.093,16.238,151.255
C08104=1106.770,387.486,-91.120,-179.090,16.243,151.255
C08105=1106.775,387.733,-91.157,-179.088,16.248,151.256
C08106=1106.781,387.981,-91.194,-179.085,16.253,151.257
C08107=1106.786,388.228,-91.231,-179.083,16.258,151.257
C08108=1106.793,388.475,-91.267,-179.080,16.262,151.258
C08109=1106.798,388.722,-91.304,-179.078,16.266,151.259
C08110=1106.803,388.969,-91.341,-179.075,16.271,151.259
C08111=1106.809,389.216,-91.379,-179.073,16.276,151.260
C08112=1106.815,389.463,-91.416,-179.070,16.281,151.260
C08113=1106.821,389.710,-91.452,-179.068,16.285,151.261
C08114=1106.827,389.958,-91.489,-179.065,16.290,151.262
C08115=1106.832,390.204,-91.526,-179.063,16.295,151.263
C08116=1106.837,390.452,-91.563,-179.060,16.300,151.263
C08117=1106.843,390.699,-91.601,-179.058,16.304,151.264
C08118=1106.850,390.946,-91.637,-179.056,16.309,151.265
C08119=1106.855,391.193,-91.674,-179.053,16.314,151.265
C08120=1106.861,391.440,-91.711,-179.051,16.319,151.266
C08121=1106.867,391.687,-91.749,-179.048,16.324,151.267
C08122=1106.872,391.934,-91.786,-179.046,16.329,151.267
C08123=1106.878,392.182,-91.823,-179.043,16.334,151.268
C08124=1106.883,392.429,-91.860,-179.041,16.339,151.269
C08125=1106.889,392.676,-91.898,-179.038,16.344,151.270
C08126=1106.894,392.923,-91.935,-179.036,16.349,151.270
C08127=1106.900,393.170,-91.972,-179.033,16.354,151.271
C08128=1106.906,393.417,-92.009,-179.032,16.358,151.272
C08129=1106.911,393.664,-92.046,-179.029,16.363,151.273
C08130=1106.917,393.911,-92.083,-179.027,16.368,151.273
C08131=1106.923,394.158,-92.121,-179.025,16.373,151.274
C08132=1106.929,394.406,-92.158,-179.022,16.379,151.275
C08133=1106.934,394.652,-92.196,-179.020,16.384,151.276
C08134=1106.940,394.900,-92.233,-179.018,16.389,151.277
C08135=1106.946,395.147,-92.270,-179.015,16.394,151.277
C08136=1106.952,395.394,-92.308,-179.013,16.399,151.278
C08137=1106.957,395.641,-92.345,-179.011,16.404,151.279
C08138=1106.963,395.888,-92.383,-179.008,16.409,151.280
C08139=1106.969,396.135,-92.420,-179.006,16.415,151.281
C08140=1106.974,396.347,-92.453,-179.004,16.420,151.281
C08141=1106.979,396.560,-92.484,-179.002,16.424,151.282
C08142=1106.983,396.772,-92.516,-179.000,16.428,151.283
C08143=1106.988,396.984,-92.549,-178.999,16.433,151.284
C08144=1106.993,397.196,-92.581,-178.996,16.437,151.284
C08145=1106.998,397.409,-92.614,-178.994,16.442,151.285
C08146=1107.002,397.621,-92.646,-178.993,16.446,151.286
C08147=1107.008,397.834,-92.678,-178.990,16.451,151.287
C08148=1107.013,398.081,-92.716,-178.988,16.456,151.287
C08149=1107.019,398.328,-92.754,-178.986,16.462,151.288
C08150=1107.024,398.575,-92.791,-178.984,16.467,151.289
C08151=1107.030,398.822,-92.829,-178.981,16.472,151.290
C08152=1107.036,399.068,-92.866,-178.979,16.478,151.291
C08153=1107.041,399.316,-92.904,-178.977,16.483,151.292
C08154=1107.047,399.563,-92.942,-178.975,16.489,151.293
C08155=1107.053,399.810,-92.980,-178.973,16.494,151.294
C08156=1107.058,400.057,-93.017,-178.970,16.500,151.295
C08157=1107.064,400.304,-93.055,-178.968,16.505,151.296
C08158=1107.070,400.551,-93.093,-178.966,16.511,151.297
C08159=1107.075,400.798,-93.132,-178.964,16.517,151.298
C08160=1107.081,401.045,-93.169,-178.962,16.522,151.298
C08161=1107.087,401.293,-93.206,-178.960,16.528,151.299
C08162=1107.092,401.540,-93.245,-178.958,16.533,151.301
C08163=1107.098,401.786,-93.282,-178.955,16.539,151.302
C08164=1107.103,402.033,-93.321,-178.953,16.545,151.302
C08165=1107.109,402.280,-93.359,-178.951,16.550,151.303
C08166=1107.115,402.527,-93.396,-178.949,16.556,151.304
C08167=1107.121,402.775,-93.435,-178.947,16.562,151.305
C08168=1107.127,403.021,-93.473,-178.944,16.568,151.306
C08169=1107.132,403.268,-93.511,-178.942,16.573,151.307
C08170=1107.137,403.516,-93.548,-178.940,16.579,151.308
C08171=1107.143,403.763,-93.586,-178.938,16.585,151.309
C08172=1107.148,404.010,-93.624,-178.936,16.590,151.310
C08173=1107.155,404.257,-93.662,-178.933,16.597,151.312
C08174=1107.160,404.504,-93.701,-178.932,16.603,151.313
C08175=1107.166,404.750,-93.739,-178.930,16.608,151.314
C08176=1107.171,404.997,-93.778,-178.928,16.614,151.315
C08177=1107.177,405.244,-93.815,-178.925,16.620,151.316
C08178=1107.183,405.492,-93.854,-178.923,16.626,151.317
C08179=1107.189,405.739,-93.892,-178.921,16.632,151.318
C08180=1107.194,405.986,-93.930,-178.919,16.638,151.319
C08181=1107.199,406.233,-93.968,-178.917,16.644,151.320
C08182=1107.205,406.479,-94.006,-178.915,16.650,151.321
C08183=1107.211,406.727,-94.045,-178.913,16.657,151.322
C08184=1107.217,406.973,-94.083,-178.911,16.662,151.323
C08185=1107.222,407.220,-94.122,-178.909,16.668,151.325
C08186=1107.228,407.467,-94.160,-178.907,16.675,151.326
C08187=1107.234,407.715,-94.198,-178.905,16.681,151.327
C08188=1107.239,407.962,-94.237,-178.903,16.687,151.328
C08189=1107.245,408.208,-94.276,-178.901,16.693,151.329
C08190=1107.251,408.455,-94.313,-178.899,16.699,151.330
C08191=1107.256,408.703,-94.352,-178.897,16.705,151.331
C08192=1107.262,408.949,-94.391,-178.895,16.712,151.333
C08193=1107.267,409.196,-94.430,-178.893,16.718,151.334
C08194=1107.273,409.443,-94.467,-178.891,16.725,151.335
C08195=1107.279,409.690,-94.507,-178.889,16.731,151.336
C08196=1107.284,409.902,-94.540,-178.887,16.737,151.337
C08197=1107.289,410.114,-94.573,-178.885,16.742,151.338
C08198=1107.293,410.327,-94.606,-178.884,16.747,151.340
C08199=1107.298,410.539,-94.639,-178.882,16.753,151.341
C08200=1107.303,410.751,-94.672,-178.880,16.759,151.342
C08201=1107.308,410.963,-94.705,-178.879,16.764,151.343
C08202=1107.312,411.175,-94.738,-178.877,16.770,151.344
C08203=1107.318,411.387,-94.772,-178.876,16.776,151.345
C08204=1107.323,411.634,-94.810,-178.874,16.782,151.346
C08205=1107.329,411.881,-94.850,-178.872,16.789,151.347
C08206=1107.334,412.128,-94.888,-178.870,16.795,151.349
C08207=1107.339,412.375,-94.927,-178.868,16.802,151.350
C08208=1107.345,412.622,-94.966,-178.867,16.808,151.351
C08209=1107.351,412.868,-95.004,-178.864,16.815,151.353
C08210=1107.357,413.116,-95.043,-178.863,16.821,151.354
C08211=1107.363,413.363,-95.082,-178.860,16.828,151.355
C08212=1107.368,413.609,-95.121,-178.858,16.835,151.356
C08213=1107.373,413.856,-95.160,-178.857,16.841,151.358
C08214=1107.379,414.103,-95.199,-178.855,16.848,151.359
C08215=1107.385,414.350,-95.237,-178.853,16.855,151.360
C08216=1107.391,414.597,-95.277,-178.851,16.862,151.362
C08217=1107.396,414.844,-95.316,-178.849,16.869,151.363
C08218=1107.402,415.090,-95.355,-178.848,16.876,151.364
C08219=1107.408,415.338,-95.393,-178.846,16.883,151.366
C08220=1107.414,415.584,-95.432,-178.844,16.889,151.367
C08221=1107.420,415.831,-95.472,-178.842,16.896,151.369
C08222=1107.425,416.078,-95.511,-178.840,16.903,151.370
C08223=1107.431,416.325,-95.550,-178.839,16.910,151.371
C08224=1107.436,416.572,-95.588,-178.837,16.917,151.373
C08225=1107.442,416.819,-95.628,-178.835,16.925,151.374
C08226=1107.448,417.066,-95.667,-178.833,16.931,151.376
C08227=1107.453,417.312,-95.706,-178.831,16.938,151.377
C08228=1107.459,417.559,-95.746,-178.829,16.946,151.379
C08229=1107.464,417.806,-95.785,-178.828,16.953,151.380
C08230=1107.470,418.053,-95.824,-178.826,16.960,151.382
C08231=1107.476,418.299,-95.864,-178.824,16.967,151.383
C08232=1107.482,418.547,-95.902,-178.823,16.975,151.384
C08233=1107.487,418.794,-95.941,-178.821,16.982,151.386
C08234=1107.492,419.040,-95.980,-178.819,16.989,151.387
C08235=1107.498,419.287,-96.020,-178.818,16.996,151.389
C08236=1107.503,419.534,-96.059,-178.816,17.004,151.390
C08237=1107.510,419.780,-96.100,-178.814,17.011,151.392
C08238=1107.515,420.027,-96.139,-178.813,17.018,151.394
C08239=1107.521,420.274,-96.178,-178.811,17.025,151.395
C08240=1107.527,420.520,-96.217,-178.809,17.033,151.397
C08241=1107.532,420.768,-96.257,-178.807,17.041,151.398
C08242=1107.537,421.014,-96.296,-178.806,17.048,151.400
C08243=1107.544,421.261,-96.336,-178.804,17.056,151.401
C08244=1107.549,421.508,-96.375,-178.803,17.063,151.403
C08245=1107.554,421.755,-96.415,-178.801,17.071,151.405
C08246=1107.560,422.001,-96.455,-178.799,17.078,151.406
C08247=1107.566,422.248,-96.494,-178.798,17.086,151.408
C08248=1107.572,422.495,-96.533,-178.796,17.093,151.409
C08249=1107.577,422.742,-96.573,-178.794,17.101,151.411
C08250=1107.583,422.989,-96.613,-178.793,17.109,151.413
C08251=1107.589,423.235,-96.652,-178.791,17.117,151.414
C08252=1107.594,423.454,-96.687,-178.790,17.123,151.416
C08253=1107.598,423.673,-96.723,-178.789,17.131,151.417
C08254=1107.604,423.891,-96.758,-178.788,17.137,151.419
C08255=1107.609,424.110,-96.793,-178.786,17.145,151.420
C08256=1107.613,424.328,-96.829,-178.784,17.151,151.422
C08257=1107.618,424.547,-96.864,-178.783,17.158,151.423
C08258=1107.624,424.766,-96.899,-178.782,17.165,151.425
C08259=1107.628,424.984,-96.934,-178.780,17.173,151.426
C08260=1107.635,425.231,-96.974,-178.779,17.181,151.428
C08261=1107.639,425.478,-97.014,-178.777,17.188,151.430
C08262=1107.646,425.724,-97.054,-178.776,17.197,151.432
C08263=1107.651,425.971,-97.093,-178.774,17.205,151.433
C08264=1107.657,426.218,-97.134,-178.773,17.213,151.435
C08265=1107.662,426.464,-97.173,-178.772,17.221,151.437
C08266=1107.668,426.711,-97.214,-178.770,17.229,151.439
C08267=1107.674,426.958,-97.253,-178.769,17.237,151.440
C08268=1107.679,427.204,-97.294,-178.767,17.245,151.442
C08269=1107.685,427.451,-97.333,-178.766,17.253,151.444
C08270=1107.691,427.698,-97.374,-178.764,17.262,151.446
C08271=1107.696,427.944,-97.414,-178.763,17.270,151.448
C08272=1107.702,428.191,-97.454,-178.762,17.278,151.450
C08273=1107.708,428.438,-97.494,-178.761,17.287,151.452
C08274=1107.713,428.684,-97.534,-178.759,17.295,151.453
C08275=1107.719,428.931,-97.574,-178.757,17.304,151.455
C08276=1107.725,429.178,-97.614,-178.756,17.312,151.457
C08277=1107.730,429.424,-97.655,-178.755,17.321,151.459
C08278=1107.736,429.670,-97.695,-178.754,17.329,151.461
C08279=1107.741,429.917,-97.734,-178.753,17.338,151.463
C08280=1107.747,430.164,-97.775,-178.751,17.346,151.465
C08281=1107.753,430.411,-97.815,-178.750,17.355,151.467
C08282=1107.758,430.657,-97.856,-178.748,17.364,151.469
C08283=1107.764,430.904,-97.896,-178.747,17.372,151.471
C08284=1107.770,431.151,-97.936,-178.746,17.381,151.473
C08285=1107.775,431.397,-97.976,-178.745,17.390,151.475
C08286=1107.781,431.644,-98.017,-178.744,17.398,151.477
C08287=1107.786,431.890,-98.058,-178.742,17.408,151.479
C08288=1107.792,432.136,-98.098,-178.741,17.416,151.481
C08289=1107.798,432.383,-98.138,-178.740,17.425,151.483
C08290=1107.803,432.630,-98.179,-178.739,17.433,151.485
C08291=1107.810,432.876,-98.219,-178.738,17.442,151.487
C08292=1107.815,433.123,-98.260,-178.736,17.452,151.489
C08293=1107.820,433.369,-98.300,-178.735,17.461,151.491
C08294=1107.826,433.616,-98.341,-178.735,17.470,151.493
C08295=1107.832,433.863,-98.382,-178.733,17.479,151.495
C08296=1107.837,434.109,-98.422,-178.732,17.488,151.497
C08297=1107.843,434.356,-98.462,-178.731,17.497,151.499
C08298=1107.849,434.602,-98.503,-178.730,17.506,151.502
C08299=1107.854,434.849,-98.543,-178.729,17.516,151.504
C08300=1107.860,435.095,-98.585,-178.728,17.525,151.506
C08301=1107.865,435.342,-98.626,-178.727,17.534,151.508
C08302=1107.870,435.588,-98.666,-178.726,17.544,151.510
C08303=1107.876,435.835,-98.707,-178.725,17.553,151.512
C08304=1107.882,436.081,-98.747,-178.724,17.563,151.515
C08305=1107.887,436.328,-98.788,-178.723,17.572,151.517
C08306=1107.893,436.574,-98.829,-178.722,17.581,151.519
C08307=1107.898,436.821,-98.870,-178.721,17.591,151.521
C08308=1107.904,437.046,-98.907,-178.720,17.600,151.523
C08309=1107.908,437.271,-98.945,-178.719,17.608,151.525
C08310=1107.914,437.496,-98.982,-178.719,17.617,151.528
C08311=1107.919,437.721,-99.019,-178.718,17.626,151.530
C08312=1107.924,437.946,-99.056,-178.717,17.635,151.532
C08313=1107.929,438.171,-99.094,-178.716,17.643,151.534
C08314=1107.934,438.396,-99.131,-178.715,17.652,151.536
C08315=1107.939,438.622,-99.169,-178.714,17.662,151.538
C08316=1107.945,438.868,-99.210,-178.713,17.671,151.540
C08317=1107.951,439.115,-99.251,-178.712,17.681,151.543
C08318=1107.957,439.361,-99.292,-178.712,17.691,151.545
C08319=1107.962,439.608,-99.333,-178.711,17.700,151.548
C08320=1107.968,439.854,-99.374,-178.710,17.710,151.550
C08321=1107.973,440.100,-99.415,-178.710,17.720,151.552
C08322=1107.979,440.346,-99.456,-178.708,17.730,151.555
C08323=1107.985,440.593,-99.497,-178.708,17.740,151.557
C08324=1107.991,440.839,-99.538,-178.707,17.751,151.560
C08325=1107.996,441.086,-99.580,-178.706,17.761,151.562
C08326=1108.002,441.333,-99.621,-178.706,17.771,151.564
C08327=1108.008,441.579,-99.663,-178.705,17.781,151.567
C08328=1108.013,441.825,-99.703,-178.704,17.791,151.570
C08329=1108.019,442.071,-99.745,-178.704,17.802,151.572
C08330=1108.024,442.318,-99.787,-178.703,17.812,151.574
C08331=1108.030,442.564,-99.827,-178.702,17.823,151.577
C08332=1108.036,442.811,-99.869,-178.701,17.833,151.580
C08333=1108.041,443.057,-99.910,-178.701,17.843,151.582
C08334=1108.046,443.304,-99.952,-178.700,17.854,151.585
C08335=1108.052,443.550,-99.993,-178.700,17.864,151.587
C08336=1108.058,443.796,-100.034,-178.699,17.875,151.590
C08337=1108.064,444.042,-100.076,-178.700,17.885,151.593
C08338=1108.069,444.288,-100.118,-178.699,17.895,151.595
C08339=1108.074,444.535,-100.158,-178.700,17.906,151.598
C08340=1108.080,444.781,-100.200,-178.700,17.917,151.601
C08341=1108.086,445.028,-100.242,-178.700,17.927,151.603
C08342=1108.092,445.274,-100.283,-178.700,17.938,151.606
C08343=1108.097,445.521,-100.325,-178.701,17.947,151.609
C08344=1108.103,445.767,-100.367,-178.701,17.958,151.612
C08345=1108.108,446.014,-100.408,-178.702,17.968,151.615
C08346=1108.114,446.260,-100.450,-178.702,17.979,151.617
C08347=1108.120,446.506,-100.491,-178.703,17.989,151.620
C08348=1108.125,446.753,-100.533,-178.705,17.999,151.623
C08349=1108.131,446.999,-100.575,-178.706,18.009,151.626
C08350=1108.136,447.246,-100.617,-178.707,18.020,151.629
C08351=1108.142,447.492,-100.658,-178.708,18.030,151.632
C08352=1108.147,447.738,-100.700,-178.709,18.041,151.635
C08353=1108.153,447.985,-100.742,-178.711,18.051,151.637
C08354=1108.158,448.231,-100.784,-178.713,18.061,151.640
C08355=1108.164,448.477,-100.825,-178.714,18.071,151.643
C08356=1108.169,448.724,-100.867,-178.716,18.081,151.646
C08357=1108.175,448.970,-100.909,-178.717,18.092,151.649
C08358=1108.181,449.217,-100.951,-178.720,18.102,151.652
C08359=1108.187,449.463,-100.992,-178.722,18.112,151.655
C08360=1108.192,449.709,-101.034,-178.723,18.122,151.658
C08361=1108.198,449.955,-101.076,-178.725,18.132,151.661
C08362=1108.203,450.202,-101.118,-178.728,18.143,151.664
C08363=1108.208,450.448,-101.160,-178.730,18.153,151.667
C08364=1107.801,450.442,-101.272,-178.813,18.385,151.743
C08365=1107.795,450.196,-101.231,-178.811,18.374,151.740
C08366=1107.790,449.950,-101.189,-178.809,18.364,151.737
C08367=1107.784,449.704,-101.147,-178.807,18.354,151.734
C08368=1107.779,449.457,-101.105,-178.805,18.344,151.731
C08369=1107.773,449.211,-101.064,-178.802,18.333,151.728
C08370=1107.767,448.964,-101.021,-178.801,18.323,151.725
C08371=1107.761,448.717,-100.980,-178.799,18.313,151.722
C08372=1107.756,448.471,-100.938,-178.798,18.302,151.719
C08373=1107.750,448.225,-100.895,-178.796,18.292,151.716
C08374=1107.744,447.979,-100.854,-178.795,18.282,151.713
C08375=1107.739,447.732,-100.812,-178.793,18.272,151.710
C08376=1107.733,447.486,-100.770,-178.791,18.261,151.707
C08377=1107.728,447.240,-100.728,-178.790,18.251,151.704
C08378=1107.722,446.993,-100.687,-178.789,18.241,151.701
C08379=1107.717,446.747,-100.645,-178.788,18.230,151.698
C08380=1107.711,446.501,-100.603,-178.787,18.220,151.695
C08381=1107.706,446.254,-100.561,-178.787,18.209,151.693
C08382=1107.700,446.008,-100.520,-178.786,18.199,151.690
C08383=1107.695,445.761,-100.478,-178.785,18.189,151.687
C08384=1107.689,445.515,-100.437,-178.784,18.178,151.684
C08385=1107.683,445.268,-100.395,-178.784,18.167,151.681
C08386=1107.678,445.022,-100.353,-178.783,18.157,151.679
C08387=1107.672,444.776,-100.312,-178.783,18.146,151.676
C08388=1107.666,444.529,-100.270,-178.783,18.136,151.673
C08389=1107.660,444.283,-100.228,-178.783,18.125,151.670
C08390=1107.655,444.037,-100.187,-178.783,18.115,151.668
C08391=1107.649,443.790,-100.145,-178.784,18.104,151.665
C08392=1107.644,443.544,-100.104,-178.784,18.094,151.662
C08393=1107.638,443.298,-100.063,-178.785,18.083,151.660
C08394=1107.633,443.051,-100.021,-178.785,18.073,151.657
C08395=1107.627,442.805,-99.979,-178.786,18.062,151.655
C08396=1107.621,442.559,-99.938,-178.787,18.051,151.652
C08397=1107.616,442.312,-99.897,-178.787,18.041,151.650
C08398=1107.610,442.066,-99.855,-178.788,18.030,151.647
C08399=1107.604,441.819,-99.814,-178.788,18.020,151.644
C08400=1107.598,441.573,-99.772,-178.789,18.010,151.642
C08401=1107.593,441.326,-99.732,-178.790,17.999,151.639
C08402=1107.587,441.081,-99.690,-178.791,17.989,151.637
C08403=1107.583,440.834,-99.649,-178.792,17.979,151.635
C08404=1107.577,440.588,-99.608,-178.792,17.969,151.632
C08405=1107.571,440.341,-99.566,-178.793,17.958,151.630
C08406=1107.565,440.095,-99.526,-178.794,17.949,151.627
C08407=1107.559,439.848,-99.484,-178.795,17.938,151.625
C08408=1107.553,439.602,-99.443,-178.796,17.928,151.622
C08409=1107.547,439.355,-99.402,-178.797,17.918,151.620
C08410=1107.542,439.109,-99.361,-178.797,17.909,151.618
C08411=1107.536,438.863,-99.320,-178.799,17.898,151.615
C08412=1107.531,438.616,-99.279,-178.799,17.889,151.613
C08413=1107.526,438.393,-99.242,-178.800,17.880,151.611
C08414=1107.520,438.169,-99.205,-178.801,17.871,151.609
C08415=1107.515,437.945,-99.167,-178.802,17.862,151.607
C08416=1107.510,437.722,-99.130,-178.803,17.853,151.604
C08417=1107.505,437.499,-99.093,-178.804,17.844,151.602
C08418=1107.500,437.275,-99.055,-178.804,17.836,151.600
C08419=1107.495,437.051,-99.018,-178.805,17.827,151.598
C08420=1107.490,436.828,-98.981,-178.806,17.818,151.596
C08421=1107.485,436.582,-98.940,-178.807,17.809,151.594
C08422=1107.479,436.335,-98.900,-178.809,17.799,151.592
C08423=1107.473,436.088,-98.859,-178.809,17.790,151.589
C08424=1107.467,435.842,-98.818,-178.811,17.780,151.587
C08425=1107.461,435.595,-98.777,-178.812,17.770,151.585
C08426=1107.456,435.349,-98.737,-178.812,17.761,151.583
C08427=1107.450,435.102,-98.696,-178.814,17.751,151.581
C08428=1107.445,434.856,-98.655,-178.815,17.742,151.578
C08429=1107.440,434.610,-98.614,-178.816,17.733,151.576
C08430=1107.434,434.363,-98.574,-178.817,17.723,151.574
C08431=1107.428,434.116,-98.533,-178.818,17.715,151.572
C08432=1107.423,433.869,-98.492,-178.819,17.705,151.570
C08433=1107.418,433.623,-98.452,-178.821,17.696,151.568
C08434=1107.412,433.377,-98.411,-178.822,17.687,151.566
C08435=1107.406,433.130,-98.371,-178.822,17.678,151.563
C08436=1107.400,432.883,-98.330,-178.824,17.668,151.561
C08437=1107.395,432.637,-98.290,-178.825,17.659,151.559
C08438=1107.389,432.390,-98.249,-178.826,17.651,151.557
C08439=1107.383,432.144,-98.209,-178.827,17.642,151.555
C08440=1107.378,431.898,-98.168,-178.829,17.633,151.553
C08441=1107.372,431.651,-98.128,-178.830,17.624,151.551
C08442=1107.366,431.404,-98.087,-178.831,17.615,151.549
C08443=1107.360,431.157,-98.047,-178.832,17.606,151.547
C08444=1107.355,430.911,-98.006,-178.834,17.597,151.545
C08445=1107.349,430.664,-97.966,-178.835,17.588,151.543
C08446=1107.344,430.418,-97.925,-178.837,17.580,151.541
C08447=1107.338,430.172,-97.885,-178.838,17.571,151.539
C08448=1107.332,429.925,-97.844,-178.839,17.562,151.537
C08449=1107.327,429.678,-97.804,-178.840,17.554,151.535
C08450=1107.321,429.432,-97.765,-178.842,17.545,151.533
C08451=1107.316,429.185,-97.724,-178.843,17.536,151.531
C08452=1107.309,428.938,-97.684,-178.844,17.528,151.530
C08453=1107.304,428.692,-97.644,-178.846,17.520,151.528
C08454=1107.299,428.445,-97.603,-178.847,17.511,151.526
C08455=1107.292,428.198,-97.563,-178.848,17.503,151.524
C08456=1107.287,427.952,-97.523,-178.850,17.495,151.522
C08457=1107.281,427.705,-97.483,-178.851,17.486,151.520
C08458=1107.276,427.458,-97.443,-178.853,17.477,151.518
C08459=1107.270,427.212,-97.404,-178.855,17.469,151.516
C08460=1107.265,426.965,-97.363,-178.856,17.461,151.515
C08461=1107.258,426.719,-97.323,-178.858,17.453,151.513
C08462=1107.253,426.472,-97.283,-178.859,17.445,151.511
C08463=1107.247,426.225,-97.243,-178.861,17.436,151.509
C08464=1107.242,425.979,-97.203,-178.862,17.428,151.507
C08465=1107.236,425.732,-97.163,-178.863,17.420,151.506
C08466=1107.231,425.485,-97.123,-178.865,17.412,151.504
C08467=1107.225,425.239,-97.083,-178.867,17.404,151.502
C08468=1107.220,424.991,-97.043,-178.868,17.396,151.501
C08469=1107.214,424.773,-97.008,-178.869,17.389,151.499
C08470=1107.209,424.554,-96.973,-178.871,17.381,151.497
C08471=1107.204,424.335,-96.937,-178.872,17.374,151.496
C08472=1107.200,424.117,-96.903,-178.873,17.368,151.494
C08473=1107.195,423.898,-96.866,-178.875,17.360,151.493
C08474=1107.189,423.679,-96.832,-178.876,17.353,151.491
C08475=1107.184,423.461,-96.796,-178.878,17.346,151.490
C08476=1107.180,423.241,-96.761,-178.879,17.339,151.488
C08477=1107.174,422.995,-96.721,-178.880,17.332,151.487
C08478=1107.168,422.748,-96.682,-178.882,17.324,151.485
C08479=1107.162,422.501,-96.642,-178.884,17.316,151.483
C08480=1107.157,422.255,-96.602,-178.885,17.308,151.482
C08481=1107.151,422.008,-96.562,-178.887,17.301,151.480
C08482=1107.145,421.761,-96.523,-178.889,17.293,151.479
C08483=1107.140,421.514,-96.483,-178.891,17.285,151.477
C08484=1107.134,421.268,-96.444,-178.892,17.277,151.475
C08485=1107.128,421.021,-96.404,-178.893,17.270,151.474
C08486=1107.122,420.775,-96.365,-178.895,17.263,151.472
C08487=1107.117,420.527,-96.325,-178.897,17.255,151.471
C08488=1107.112,420.281,-96.286,-178.899,17.247,151.469
C08489=1107.106,420.034,-96.247,-178.901,17.240,151.467
C08490=1107.100,419.787,-96.208,-178.902,17.232,151.466
C08491=1107.094,419.541,-96.167,-178.904,17.226,151.464
C08492=1107.089,419.294,-96.128,-178.905,17.218,151.463
C08493=1107.083,419.047,-96.088,-178.907,17.210,151.461
C08494=1107.077,418.800,-96.049,-178.909,17.203,151.460
C08495=1107.071,418.553,-96.010,-178.911,17.195,151.458
C08496=1107.066,418.307,-95.971,-178.912,17.189,151.457
C08497=1107.060,418.060,-95.931,-178.914,17.181,151.455
C08498=1107.055,417.813,-95.892,-178.916,17.174,151.454
C08499=1107.049,417.566,-95.852,-178.918,17.166,151.452
C08500=1107.044,417.319,-95.814,-178.920,17.160,151.451
C08501=1107.038,417.072,-95.775,-178.921,17.152,151.449
C08502=1107.032,416.825,-95.735,-178.923,17.145,151.448
C08503=1107.027,416.579,-95.696,-178.925,17.138,151.446
C08504=1107.021,416.332,-95.657,-178.927,17.131,151.445
C08505=1107.015,416.085,-95.618,-178.929,17.124,151.444
C08506=1107.009,415.838,-95.578,-178.931,17.117,151.442
C08507=1107.004,415.591,-95.540,-178.932,17.110,151.441
C08508=1106.998,415.344,-95.501,-178.934,17.103,151.439
C08509=1106.993,415.097,-95.462,-178.937,17.096,151.438
C08510=1106.986,414.850,-95.422,-178.938,17.089,151.437
C08511=1106.981,414.604,-95.383,-178.940,17.082,151.435
C08512=1106.976,414.357,-95.345,-178.942,17.076,151.434
C08513=1106.970,414.110,-95.305,-178.944,17.068,151.433
C08514=1106.964,413.863,-95.267,-178.946,17.061,151.431
C08515=1106.958,413.616,-95.228,-178.947,17.055,151.430
C08516=1106.952,413.369,-95.189,-178.949,17.048,151.429
C08517=1106.947,413.123,-95.150,-178.951,17.042,151.427
C08518=1106.941,412.875,-95.111,-178.953,17.035,151.426
C08519=1106.936,412.629,-95.072,-178.955,17.028,151.425
C08520=1106.930,412.382,-95.034,-178.957,17.021,151.423
C08521=1106.924,412.134,-94.994,-178.959,17.014,151.422
C08522=1106.918,411.888,-94.956,-178.961,17.008,151.421
C08523=1106.912,411.641,-94.917,-178.963,17.001,151.420
C08524=1106.907,411.394,-94.878,-178.965,16.995,151.418
C08525=1106.902,411.182,-94.845,-178.966,16.989,151.417
C08526=1106.898,410.970,-94.812,-178.968,16.983,151.416
C08527=1106.893,410.757,-94.779,-178.969,16.978,151.415
C08528=1106.888,410.545,-94.745,-178.971,16.972,151.414
C08529=1106.883,410.332,-94.712,-178.973,16.966,151.413
C08530=1106.878,410.120,-94.679,-178.975,16.961,151.412
C08531=1106.874,409.908,-94.646,-178.976,16.955,151.411
C08532=1106.869,409.696,-94.613,-178.978,16.950,151.410
C08533=1106.863,409.449,-94.573,-178.980,16.944,151.408
C08534=1106.857,409.202,-94.535,-178.982,16.937,151.407
C08535=1106.852,408.955,-94.497,-178.984,16.931,151.406
C08536=1106.846,408.708,-94.458,-178.986,16.924,151.405
C08537=1106.841,408.461,-94.420,-178.988,16.918,151.404
C08538=1106.834,408.214,-94.381,-178.991,16.911,151.402
C08539=1106.829,407.968,-94.342,-178.992,16.905,151.401
C08540=1106.824,407.720,-94.304,-178.994,16.899,151.400
C08541=1106.817,407.473,-94.266,-178.997,16.893,151.399
C08542=1106.812,407.226,-94.228,-178.998,16.887,151.398
C08543=1106.807,406.980,-94.189,-179.001,16.880,151.397
C08544=1106.801,406.733,-94.151,-179.003,16.874,151.395
C08545=1106.796,406.486,-94.112,-179.004,16.868,151.394
C08546=1106.790,406.238,-94.074,-179.007,16.862,151.393
C08547=1106.784,405.991,-94.036,-179.009,16.856,151.392
C08548=1106.779,405.744,-93.998,-179.010,16.850,151.391
C08549=1106.773,405.498,-93.959,-179.013,16.844,151.390
C08550=1106.767,405.250,-93.920,-179.015,16.838,151.389
C08551=1106.761,405.004,-93.883,-179.017,16.832,151.388
C08552=1106.756,404.756,-93.844,-179.019,16.826,151.387
C08553=1106.750,404.510,-93.807,-179.022,16.820,151.386
C08554=1106.745,404.263,-93.768,-179.023,16.814,151.384
C08555=1106.738,404.015,-93.730,-179.025,16.808,151.383
C08556=1106.733,403.768,-93.692,-179.028,16.802,151.382
C08557=1106.727,403.521,-93.654,-179.030,16.796,151.381
C08558=1106.722,403.274,-93.616,-179.032,16.790,151.380
C08559=1106.716,403.028,-93.578,-179.034,16.785,151.379
C08560=1106.710,402.780,-93.539,-179.037,16.778,151.378
C08561=1106.704,402.533,-93.501,-179.039,16.773,151.377
C08562=1106.699,402.286,-93.463,-179.041,16.767,151.376
C08563=1106.693,402.039,-93.425,-179.043,16.762,151.375
C08564=1106.687,401.793,-93.388,-179.045,16.756,151.374
C08565=1106.682,401.546,-93.349,-179.047,16.750,151.373
C08566=1106.677,401.298,-93.312,-179.049,16.744,151.372
C08567=1106.671,401.050,-93.273,-179.051,16.738,151.371
C08568=1106.665,400.804,-93.236,-179.053,16.733,151.370
C08569=1106.659,400.557,-93.198,-179.055,16.727,151.369
C08570=1106.654,400.310,-93.160,-179.058,16.722,151.368
C08571=1106.648,400.062,-93.123,-179.061,16.716,151.367
C08572=1106.642,399.816,-93.085,-179.063,16.710,151.366
C08573=1106.637,399.569,-93.046,-179.065,16.705,151.366
C08574=1106.631,399.322,-93.009,-179.067,16.699,151.365
C08575=1106.626,399.075,-92.972,-179.069,16.694,151.364
C08576=1106.620,398.828,-92.934,-179.071,16.688,151.363
C08577=1106.614,398.580,-92.895,-179.073,16.683,151.362
C08578=1106.608,398.333,-92.857,-179.075,16.678,151.361
C08579=1106.603,398.086,-92.820,-179.078,16.672,151.360
C08580=1106.597,397.839,-92.783,-179.080,16.667,151.359
C08581=1106.592,397.626,-92.750,-179.082,16.662,151.358
C08582=1106.587,397.414,-92.717,-179.084,16.658,151.358
C08583=1106.582,397.202,-92.686,-179.086,16.652,151.357
C08584=1106.577,396.989,-92.653,-179.088,16.648,151.356
C08585=1106.573,396.776,-92.621,-179.090,16.644,151.355
C08586=1106.567,396.565,-92.589,-179.092,16.639,151.355
C08587=1106.563,396.353,-92.557,-179.094,16.634,151.354
C08588=1106.559,396.140,-92.524,-179.096,16.630,151.353
C08589=1106.553,395.893,-92.487,-179.098,16.625,151.352
C08590=1106.547,395.646,-92.450,-179.100,16.620,151.351
C08591=1106.541,395.399,-92.412,-179.103,16.614,151.351
C08592=1106.536,395.152,-92.375,-179.105,16.609,151.350
C08593=1106.530,394.905,-92.337,-179.107,16.604,151.349
C08594=1106.524,394.658,-92.300,-179.109,16.599,151.348
C08595=1106.519,394.410,-92.262,-179.112,16.594,151.347
C08596=1106.513,394.163,-92.225,-179.114,16.589,151.347
C08597=1106.507,393.916,-92.187,-179.117,16.583,151.346
C08598=1106.502,393.669,-92.150,-179.119,16.578,151.345
C08599=1106.496,393.422,-92.113,-179.121,16.573,151.344
C08600=1106.490,393.175,-92.075,-179.124,16.568,151.343
C08601=1106.485,392.927,-92.038,-179.126,16.563,151.343
C08602=1106.479,392.680,-92.001,-179.129,16.558,151.342
C08603=1106.473,392.433,-91.963,-179.131,16.553,151.341
C08604=1106.468,392.186,-91.926,-179.133,16.548,151.340
C08605=1106.461,391.939,-91.890,-179.136,16.543,151.340
C08606=1106.455,391.692,-91.852,-179.138,16.538,151.339
C08607=1106.450,391.445,-91.815,-179.141,16.533,151.338
C08608=1106.445,391.198,-91.778,-179.143,16.528,151.337
C08609=1106.439,390.951,-91.741,-179.146,16.523,151.337
C08610=1106.433,390.704,-91.704,-179.149,16.518,151.336
C08611=1106.428,390.457,-91.667,-179.151,16.513,151.335
C08612=1106.421,390.210,-91.630,-179.153,16.509,151.334
C08613=1106.416,389.962,-91.593,-179.155,16.504,151.334
C08614=1106.410,389.716,-91.555,-179.158,16.499,151.333
C08615=1106.404,389.468,-91.518,-179.160,16.494,151.332
C08616=1106.399,389.222,-91.482,-179.163,16.489,151.332
C08617=1106.393,388.974,-91.445,-179.165,16.485,151.331
C08618=1106.387,388.727,-91.408,-179.168,16.480,151.330
C08619=1106.382,388.480,-91.371,-179.171,16.475,151.330
C08620=1106.376,388.232,-91.334,-179.173,16.470,151.329
C08621=1106.370,387.985,-91.298,-179.175,16.466,151.329
C08622=1106.365,387.739,-91.261,-179.178,16.461,151.328
C08623=1106.359,387.491,-91.224,-179.180,16.456,151.327
C08624=1106.354,387.244,-91.187,-179.183,16.452,151.326
C08625=1106.347,386.997,-91.150,-179.186,16.447,151.326
C08626=1106.342,386.750,-91.113,-179.188,16.442,151.325
C08627=1106.337,386.503,-91.077,-179.191,16.437,151.325
C08628=1106.330,386.256,-91.040,-179.193,16.433,151.324
C08629=1106.325,386.008,-91.003,-179.196,16.429,151.323
C08630=1106.319,385.761,-90.966,-179.198,16.424,151.323
C08631=1106.314,385.514,-90.929,-179.201,16.419,151.322
C08632=1106.308,385.267,-90.893,-179.204,16.414,151.321
C08633=1106.302,385.020,-90.856,-179.206,16.410,151.321
C08634=1106.297,384.773,-90.819,-179.208,16.406,151.320
C08635=1106.291,384.526,-90.783,-179.211,16.401,151.320
C08636=1106.286,384.278,-90.747,-179.214,16.396,151.319
C08637=1106.276,383.866,-90.685,-179.218,16.389,151.318
C08638=1106.266,383.453,-90.625,-179.222,16.382,151.317
C08639=1106.257,383.041,-90.563,-179.227,16.374,151.316
C08640=1106.248,382.628,-90.502,-179.231,16.367,151.315
C08641=1106.242,382.380,-90.466,-179.234,16.362,151.315
C08642=1106.237,382.133,-90.429,-179.236,16.358,151.314
C08643=1106.231,381.886,-90.393,-179.239,16.354,151.314
C08644=1106.225,381.639,-90.357,-179.242,16.349,151.313
C08645=1106.219,381.391,-90.320,-179.245,16.345,151.313
C08646=1106.213,381.145,-90.284,-179.247,16.341,151.312
C08647=1106.208,380.897,-90.248,-179.250,16.337,151.312
C08648=1106.202,380.650,-90.211,-179.252,16.332,151.311
C08649=1106.197,380.403,-90.175,-179.255,16.329,151.311
C08650=1106.191,380.156,-90.139,-179.258,16.324,151.310
C08651=1106.184,379.909,-90.102,-179.261,16.320,151.310
C08652=1106.180,379.661,-90.066,-179.263,16.316,151.309
C08653=1106.173,379.414,-90.030,-179.265,16.311,151.309
C08654=1106.168,379.166,-89.994,-179.269,16.307,151.308
C08655=1106.162,378.920,-89.958,-179.271,16.303,151.308
C08656=1106.156,378.672,-89.922,-179.274,16.299,151.307
C08657=1106.151,378.425,-89.885,-179.276,16.295,151.307
C08658=1106.145,378.178,-89.849,-179.280,16.290,151.306
C08659=1106.140,377.930,-89.813,-179.282,16.287,151.306
C08660=1106.134,377.684,-89.777,-179.285,16.283,151.306
C08661=1106.128,377.436,-89.741,-179.288,16.278,151.305
C08662=1106.123,377.189,-89.704,-179.290,16.274,151.304
C08663=1106.117,376.942,-89.669,-179.293,16.270,151.304
C08664=1106.111,376.694,-89.633,-179.295,16.266,151.304
C08665=1106.106,376.447,-89.597,-179.298,16.262,151.303
C08666=1106.100,376.200,-89.561,-179.301,16.258,151.303
C08667=1106.095,375.953,-89.525,-179.303,16.254,151.302
C08668=1106.088,375.706,-89.489,-179.306,16.250,151.302
C08669=1106.084,375.458,-89.453,-179.309,16.246,151.301
C08670=1106.078,375.211,-89.417,-179.312,16.242,151.301
C08671=1106.072,374.963,-89.382,-179.315,16.238,151.301
C08672=1106.067,374.716,-89.345,-179.317,16.234,151.300
C08673=1106.060,374.469,-89.309,-179.320,16.230,151.300
C08674=1106.055,374.222,-89.274,-179.323,16.226,151.300
C08675=1106.049,373.974,-89.238,-179.326,16.223,151.299
C08676=1106.044,373.727,-89.203,-179.329,16.219,151.299
C08677=1106.037,373.480,-89.166,-179.331,16.215,151.298
C08678=1106.032,373.232,-89.130,-179.334,16.211,151.298
C08679=1106.027,372.985,-89.095,-179.337,16.208,151.298
C08680=1106.020,372.737,-89.059,-179.340,16.204,151.297
C08681=1106.015,372.490,-89.023,-179.343,16.199,151.297
C08682=1106.009,372.243,-88.988,-179.345,16.196,151.297
C08683=1106.004,371.996,-88.952,-179.349,16.192,151.296
C08684=1105.998,371.748,-88.917,-179.351,16.188,151.296
C08685=1105.992,371.501,-88.881,-179.354,16.184,151.296
C08686=1105.986,371.253,-88.846,-179.356,16.181,151.295
C08687=1105.981,371.006,-88.810,-179.360,16.177,151.295
C08688=1105.975,370.759,-88.774,-179.362,16.174,151.295
C08689=1105.967,370.373,-88.719,-179.367,16.168,151.294
C08690=1105.957,369.987,-88.663,-179.371,16.162,151.294
C08691=1105.948,369.601,-88.608,-179.376,16.156,151.293
C08692=1105.940,369.215,-88.552,-179.381,16.150,151.293
C08693=1105.934,368.967,-88.516,-179.383,16.147,151.292
C08694=1105.929,368.720,-88.482,-179.386,16.143,151.292
C08695=1105.923,368.472,-88.446,-179.389,16.140,151.292
C08696=1105.917,368.225,-88.411,-179.392,16.135,151.291
C08697=1105.912,367.978,-88.375,-179.395,16.132,151.291
C08698=1105.906,367.730,-88.340,-179.398,16.128,151.291
C08699=1105.900,367.483,-88.306,-179.401,16.125,151.291
C08700=1105.894,367.235,-88.270,-179.403,16.122,151.290
C08701=1105.889,366.988,-88.235,-179.406,16.118,151.290
C08702=1105.883,366.741,-88.199,-179.409,16.115,151.290
C08703=1105.877,366.493,-88.164,-179.412,16.111,151.290
C08704=1105.872,366.246,-88.129,-179.415,16.108,151.289
C08705=1105.866,365.999,-88.093,-179.418,16.104,151.289
C08706=1105.861,365.751,-88.058,-179.421,16.101,151.289
C08707=1105.855,365.504,-88.023,-179.424,16.097,151.289
C08708=1105.849,365.256,-87.987,-179.427,16.094,151.288
C08709=1105.844,365.009,-87.953,-179.430,16.090,151.288
C08710=1105.838,364.761,-87.918,-179.433,16.087,151.288
C08711=1105.832,364.514,-87.882,-179.435,16.083,151.288
C08712=1105.827,364.267,-87.848,-179.438,16.080,151.287
C08713=1105.821,364.019,-87.812,-179.441,16.077,151.287
C08714=1105.815,363.772,-87.778,-179.445,16.073,151.287
C08715=1105.809,363.524,-87.742,-179.447,16.070,151.287
C08716=1105.804,363.277,-87.707,-179.451,16.066,151.287
C08717=1105.798,363.030,-87.672,-179.453,16.063,151.286
C08718=1105.792,362.782,-87.638,-179.456,16.060,151.286
C08719=1105.787,362.535,-87.602,-179.460,16.056,151.286
C08720=1105.781,362.287,-87.568,-179.462,16.053,151.286
C08721=1105.775,362.040,-87.532,-179.465,16.050,151.286
C08722=1105.770,361.792,-87.498,-179.468,16.046,151.286
C08723=1105.764,361.545,-87.462,-179.471,16.043,151.285
C08724=1105.758,361.297,-87.428,-179.474,16.040,151.285
C08725=1105.753,361.050,-87.393,-179.477,16.037,151.285
C08726=1105.747,360.803,-87.358,-179.480,16.034,151.285
C08727=1105.741,360.554,-87.323,-179.483,16.030,151.285
C08728=1105.736,360.307,-87.289,-179.486,16.027,151.284
C08729=1105.730,360.060,-87.254,-179.489,16.024,151.284
C08730=1105.724,359.813,-87.220,-179.492,16.020,151.284
C08731=1105.719,359.564,-87.184,-179.495,16.017,151.284
C08732=1105.712,359.318,-87.150,-179.499,16.014,151.284
C08733=1105.707,359.070,-87.115,-179.502,16.011,151.284
C08734=1105.702,358.822,-87.080,-179.504,16.008,151.284
C08735=1105.696,358.575,-87.046,-179.508,16.005,151.284
C08736=1105.690,358.328,-87.011,-179.511,16.002,151.283
C08737=1105.684,358.080,-86.976,-179.513,15.999,151.283
C08738=1105.679,357.832,-86.942,-179.517,15.995,151.283
C08739=1105.673,357.585,-86.908,-179.520,15.992,151.283
C08740=1105.668,357.337,-86.873,-179.523,15.989,151.283
C08741=1105.659,356.966,-86.820,-179.528,15.984,151.283
C08742=1105.650,356.595,-86.769,-179.532,15.980,151.283
C08743=1105.642,356.223,-86.718,-179.537,15.975,151.282
C08744=1105.634,355.852,-86.666,-179.541,15.971,151.282
C08745=1105.627,355.604,-86.631,-179.544,15.968,151.282
C08746=1105.622,355.357,-86.597,-179.548,15.965,151.282
C08747=1105.616,355.110,-86.563,-179.550,15.962,151.282
C08748=1105.611,354.862,-86.529,-179.553,15.959,151.282
C08749=1105.605,354.615,-86.494,-179.556,15.956,151.282
C08750=1105.599,354.367,-86.459,-179.560,15.953,151.282
C08751=1105.594,354.119,-86.425,-179.563,15.950,151.282
C08752=1105.588,353.872,-86.391,-179.566,15.947,151.282
C08753=1105.583,353.624,-86.356,-179.569,15.943,151.281
C08754=1105.577,353.377,-86.322,-179.572,15.941,151.281
C08755=1105.571,353.129,-86.288,-179.575,15.938,151.281
C08756=1105.565,352.881,-86.253,-179.578,15.936,151.281
C08757=1105.560,352.634,-86.219,-179.582,15.932,151.281
C08758=1105.554,352.386,-86.186,-179.585,15.930,151.281
C08759=1105.548,352.139,-86.152,-179.588,15.926,151.281
C08760=1105.543,351.891,-86.117,-179.591,15.924,151.281
C08761=1105.537,351.643,-86.082,-179.594,15.921,151.281
C08762=1105.531,351.396,-86.048,-179.597,15.918,151.281
C08763=1105.526,351.148,-86.014,-179.600,15.915,151.281
C08764=1105.520,350.901,-85.980,-179.603,15.913,151.281
C08765=1105.514,350.653,-85.946,-179.606,15.910,151.281
C08766=1105.508,350.406,-85.912,-179.610,15.907,151.281
C08767=1105.503,350.158,-85.878,-179.613,15.904,151.281
C08768=1105.498,349.910,-85.844,-179.616,15.901,151.281
C08769=1105.491,349.662,-85.810,-179.619,15.899,151.281
C08770=1105.485,349.415,-85.776,-179.622,15.896,151.281
C08771=1105.480,349.167,-85.743,-179.626,15.893,151.281
C08772=1105.475,348.920,-85.708,-179.629,15.890,151.281
C08773=1105.469,348.672,-85.674,-179.632,15.888,151.281
C08774=1105.463,348.425,-85.640,-179.635,15.885,151.281
C08775=1105.457,348.177,-85.606,-179.638,15.882,151.281
C08776=1105.452,347.929,-85.573,-179.642,15.879,151.281
C08777=1105.446,347.682,-85.539,-179.645,15.876,151.281
C08778=1105.441,347.434,-85.505,-179.648,15.874,151.281
C08779=1105.435,347.187,-85.471,-179.651,15.871,151.281
C08780=1105.429,346.939,-85.437,-179.654,15.869,151.281
C08781=1105.424,346.691,-85.404,-179.657,15.866,151.281
C08782=1105.417,346.443,-85.369,-179.661,15.863,151.281
C08783=1105.412,346.195,-85.336,-179.664,15.860,151.281
C08784=1105.406,345.948,-85.303,-179.667,15.858,151.281
C08785=1105.400,345.700,-85.269,-179.670,15.855,151.281
C08786=1105.395,345.452,-85.235,-179.673,15.853,151.281
C08787=1105.389,345.205,-85.201,-179.676,15.850,151.281
C08788=1105.383,344.957,-85.168,-179.679,15.848,151.281
C08789=1105.378,344.710,-85.134,-179.683,15.845,151.281
C08790=1105.372,344.462,-85.100,-179.686,15.842,151.281
C08791=1105.366,344.214,-85.067,-179.690,15.840,151.282
C08792=1105.361,343.967,-85.033,-179.693,15.837,151.282
C08793=1105.352,343.598,-84.983,-179.697,15.833,151.282
C08794=1105.344,343.228,-84.934,-179.702,15.830,151.282
C08795=1105.335,342.860,-84.883,-179.707,15.826,151.282
C08796=1105.327,342.491,-84.833,-179.712,15.823,151.282
C08797=1105.321,342.243,-84.800,-179.716,15.819,151.282
C08798=1105.316,341.995,-84.767,-179.719,15.817,151.282
C08799=1105.310,341.747,-84.733,-179.722,15.814,151.282
C08800=1105.304,341.500,-84.699,-179.725,15.812,151.282
C08801=1105.299,341.252,-84.666,-179.729,15.810,151.283
C08802=1105.293,341.004,-84.633,-179.732,15.807,151.283
C08803=1105.287,340.756,-84.600,-179.735,15.805,151.283
C08804=1105.281,340.508,-84.566,-179.738,15.803,151.283
C08805=1105.276,340.261,-84.532,-179.741,15.800,151.283
C08806=1105.270,340.013,-84.499,-179.744,15.798,151.283
C08807=1105.265,339.766,-84.466,-179.748,15.796,151.283
C08808=1105.260,339.518,-84.433,-179.751,15.793,151.283
C08809=1105.253,339.271,-84.400,-179.755,15.790,151.283
C08810=1105.248,339.023,-84.367,-179.758,15.788,151.283
C08811=1105.242,338.775,-84.333,-179.761,15.785,151.284
C08812=1105.237,338.527,-84.300,-179.765,15.783,151.284
C08813=1105.231,338.279,-84.267,-179.768,15.781,151.284
C08814=1105.225,338.031,-84.234,-179.771,15.778,151.284
C08815=1105.219,337.783,-84.201,-179.774,15.776,151.284
C08816=1105.214,337.536,-84.167,-179.778,15.774,151.284
C08817=1105.207,337.288,-84.135,-179.781,15.771,151.284
C08818=1105.202,337.041,-84.102,-179.784,15.769,151.284
C08819=1105.197,336.793,-84.068,-179.787,15.767,151.285
C08820=1105.191,336.545,-84.035,-179.791,15.765,151.285
C08821=1105.185,336.297,-84.002,-179.794,15.762,151.285
C08822=1105.179,336.049,-83.969,-179.797,15.760,151.285
C08823=1105.173,335.801,-83.937,-179.801,15.758,151.285
C08824=1105.168,335.553,-83.903,-179.804,15.756,151.285
C08825=1105.163,335.306,-83.870,-179.807,15.753,151.286
C08826=1105.157,335.058,-83.838,-179.811,15.751,151.286
C08827=1105.151,334.811,-83.804,-179.814,15.749,151.286
C08828=1105.146,334.563,-83.771,-179.817,15.747,151.286
C08829=1105.140,334.314,-83.739,-179.820,15.744,151.286
C08830=1105.135,334.067,-83.706,-179.824,15.742,151.286
C08831=1105.128,333.820,-83.673,-179.827,15.740,151.287
C08832=1105.123,333.572,-83.640,-179.831,15.738,151.287
C08833=1105.117,333.323,-83.607,-179.834,15.736,151.287
C08834=1105.111,333.076,-83.575,-179.837,15.733,151.287
C08835=1105.106,332.828,-83.542,-179.841,15.731,151.287
C08836=1105.100,332.580,-83.510,-179.844,15.729,151.287
C08837=1105.095,332.332,-83.476,-179.847,15.727,151.288
C08838=1105.088,332.085,-83.444,-179.851,15.725,151.288
C08839=1105.083,331.836,-83.411,-179.854,15.723,151.288
C08840=1105.077,331.589,-83.379,-179.857,15.720,151.288
C08841=1105.072,331.341,-83.345,-179.861,15.718,151.288
C08842=1105.066,331.093,-83.313,-179.864,15.716,151.289
C08843=1105.060,330.846,-83.280,-179.867,15.715,151.289
C08844=1105.054,330.598,-83.247,-179.871,15.713,151.289
C08845=1105.045,330.223,-83.198,-179.876,15.710,151.289
C08846=1105.037,329.848,-83.149,-179.881,15.706,151.290
C08847=1105.028,329.472,-83.100,-179.886,15.703,151.290
C08848=1105.019,329.097,-83.050,-179.891,15.700,151.291
C08849=1105.013,328.849,-83.018,-179.895,15.698,151.291
C08850=1105.008,328.602,-82.987,-179.898,15.696,151.291
C08851=1105.002,328.354,-82.953,-179.901,15.694,151.291
C08852=1104.996,328.105,-82.921,-179.905,15.692,151.292
C08853=1104.990,327.858,-82.889,-179.908,15.690,151.292
C08854=1104.985,327.610,-82.856,-179.912,15.688,151.292
C08855=1104.979,327.362,-82.824,-179.915,15.686,151.292
C08856=1104.973,327.114,-82.791,-179.918,15.685,151.292
C08857=1104.967,326.866,-82.759,-179.922,15.682,151.293
C08858=1104.962,326.619,-82.726,-179.925,15.681,151.293
C08859=1104.956,326.371,-82.694,-179.929,15.679,151.293
C08860=1104.950,326.122,-82.662,-179.932,15.676,151.293
C08861=1104.944,325.875,-82.630,-179.936,15.675,151.294
C08862=1104.939,325.627,-82.597,-179.939,15.672,151.294
C08863=1104.933,325.379,-82.565,-179.942,15.671,151.294
C08864=1104.928,325.132,-82.533,-179.945,15.669,151.295
C08865=1104.922,324.884,-82.501,-179.949,15.667,151.295
C08866=1104.917,324.636,-82.469,-179.952,15.665,151.295
C08867=1104.911,324.388,-82.437,-179.956,15.663,151.295
C08868=1104.905,324.139,-82.405,-179.959,15.661,151.296
C08869=1104.899,323.892,-82.372,-179.963,15.659,151.296
C08870=1104.893,323.644,-82.340,-179.967,15.657,151.296
C08871=1104.888,323.397,-82.309,-179.969,15.656,151.296
C08872=1104.883,323.148,-82.276,-179.973,15.654,151.297
C08873=1104.877,322.900,-82.244,-179.976,15.652,151.297
C08874=1104.871,322.652,-82.212,-179.980,15.650,151.297
C08875=1104.865,322.405,-82.180,-179.983,15.648,151.297
C08876=1104.860,322.157,-82.148,-179.987,15.646,151.298
C08877=1104.854,321.909,-82.116,-179.990,15.645,151.298
C08878=1104.849,321.661,-82.084,-179.993,15.643,151.298
C08879=1104.843,321.413,-82.052,-179.997,15.641,151.299
C08880=1104.837,321.165,-82.020,180.000,15.639,151.299
C08881=1104.832,320.917,-81.988,179.996,15.637,151.299
C08882=1104.826,320.669,-81.956,179.993,15.635,151.299
C08883=1104.820,320.422,-81.924,179.990,15.634,151.300
C08884=1104.814,320.173,-81.892,179.986,15.632,151.300
C08885=1104.809,319.926,-81.861,179.983,15.630,151.300
C08886=1104.803,319.678,-81.829,179.979,15.628,151.301
C08887=1104.797,319.430,-81.797,179.976,15.626,151.301
C08888=1104.791,319.182,-81.765,179.972,15.624,151.301
C08889=1104.786,318.934,-81.733,179.969,15.623,151.302
C08890=1104.781,318.687,-81.702,179.966,15.621,151.302
C08891=1104.776,318.438,-81.670,179.962,15.619,151.302
C08892=1104.770,318.190,-81.638,179.958,15.617,151.303
C08893=1104.764,317.942,-81.606,179.955,15.615,151.303
C08894=1104.759,317.695,-81.574,179.952,15.614,151.303
C08895=1104.753,317.446,-81.542,179.949,15.612,151.303
C08896=1104.748,317.199,-81.511,179.945,15.610,151.304
C08897=1104.739,316.816,-81.463,179.940,15.607,151.304
C08898=1104.730,316.435,-81.414,179.934,15.605,151.305
C08899=1104.722,316.052,-81.364,179.929,15.603,151.305
C08900=1104.713,315.670,-81.316,179.924,15.600,151.306
C08901=1104.707,315.422,-81.284,179.920,15.598,151.306
C08902=1104.702,315.174,-81.253,179.917,15.596,151.306
C08903=1104.696,314.925,-81.221,179.913,15.595,151.307
C08904=1104.690,314.678,-81.190,179.910,15.593,151.307
C08905=1104.684,314.430,-81.158,179.906,15.592,151.307
C08906=1104.679,314.182,-81.127,179.903,15.590,151.308
C08907=1104.672,313.934,-81.096,179.899,15.588,151.308
C08908=1104.667,313.686,-81.064,179.896,15.587,151.309
C08909=1104.662,313.438,-81.033,179.892,15.585,151.309
C08910=1104.655,313.190,-81.002,179.889,15.583,151.309
C08911=1104.650,312.943,-80.970,179.885,15.582,151.310
C08912=1104.644,312.694,-80.939,179.882,15.581,151.310
C08913=1104.638,312.447,-80.908,179.878,15.579,151.310
C08914=1104.633,312.199,-80.877,179.874,15.578,151.311
C08915=1104.627,311.950,-80.845,179.871,15.576,151.311
C08916=1104.621,311.703,-80.814,179.868,15.575,151.312
C08917=1104.615,311.454,-80.782,179.864,15.573,151.312
C08918=1104.610,311.207,-80.751,179.860,15.571,151.312
C08919=1104.604,310.959,-80.720,179.857,15.570,151.313
C08920=1104.598,310.711,-80.688,179.853,15.569,151.313
C08921=1104.592,310.463,-80.658,179.850,15.567,151.314
C08922=1104.587,310.215,-80.627,179.846,15.565,151.314
C08923=1104.581,309.967,-80.595,179.843,15.564,151.314
C08924=1104.575,309.719,-80.565,179.839,15.562,151.315
C08925=1104.570,309.471,-80.533,179.836,15.561,151.315
C08926=1104.563,309.223,-80.502,179.833,15.560,151.316
C08927=1104.558,308.975,-80.471,179.829,15.558,151.316
C08928=1104.552,308.727,-80.440,179.825,15.557,151.316
C08929=1104.547,308.479,-80.409,179.822,15.555,151.317
C08930=1104.540,308.231,-80.378,179.818,15.554,151.317
C08931=1104.535,307.983,-80.347,179.815,15.552,151.318
C08932=1104.530,307.735,-80.317,179.811,15.550,151.318
C08933=1104.524,307.487,-80.285,179.808,15.549,151.318
C08934=1104.519,307.239,-80.254,179.804,15.548,151.319
C08935=1104.513,306.991,-80.223,179.800,15.546,151.319
C08936=1104.508,306.743,-80.192,179.797,15.545,151.320
C08937=1104.501,306.495,-80.161,179.793,15.544,151.320
C08938=1104.495,306.247,-80.131,179.790,15.542,151.320
C08939=1104.490,305.999,-80.100,179.786,15.540,151.321
C08940=1104.484,305.751,-80.069,179.783,15.539,151.321
C08941=1104.479,305.503,-80.038,179.779,15.538,151.322
C08942=1104.472,305.255,-80.007,179.775,15.536,151.322
C08943=1104.467,305.007,-79.976,179.772,15.535,151.323
C08944=1104.461,304.759,-79.946,179.769,15.533,151.323
C08945=1104.456,304.511,-79.915,179.765,15.532,151.324
C08946=1104.451,304.264,-79.884,179.762,15.531,151.324
C08947=1104.445,304.015,-79.853,179.758,15.529,151.324
C08948=1104.440,303.768,-79.823,179.754,15.527,151.325
C08949=1104.430,303.388,-79.776,179.749,15.526,151.325
C08950=1104.422,303.008,-79.729,179.743,15.523,151.326
C08951=1104.413,302.629,-79.682,179.738,15.521,151.327
C08952=1104.405,302.248,-79.635,179.733,15.519,151.327
C08953=1104.399,302.001,-79.605,179.729,15.518,151.328
C08954=1104.394,301.752,-79.574,179.725,15.516,151.328
C08955=1104.388,301.505,-79.543,179.722,15.515,151.329
C08956=1104.383,301.257,-79.513,179.718,15.514,151.329
C08957=1104.377,301.009,-79.482,179.714,15.512,151.330
C08958=1104.372,300.761,-79.452,179.711,15.511,151.330
C08959=1104.366,300.513,-79.421,179.708,15.510,151.330
C08960=1104.360,300.264,-79.390,179.704,15.509,151.331
C08961=1104.354,300.016,-79.360,179.700,15.507,151.331
C08962=1104.348,299.769,-79.329,179.697,15.506,151.332
C08963=1104.344,299.520,-79.299,179.694,15.505,151.332
C08964=1104.338,299.272,-79.269,179.690,15.503,151.333
C08965=1104.332,299.024,-79.238,179.686,15.502,151.333
C08966=1104.326,298.776,-79.208,179.683,15.501,151.334
C08967=1104.321,298.528,-79.177,179.679,15.499,151.334
C08968=1104.315,298.280,-79.147,179.675,15.498,151.334
C08969=1104.310,298.032,-79.117,179.672,15.497,151.335
C08970=1104.304,297.784,-79.087,179.668,15.495,151.335
C08971=1104.298,297.536,-79.056,179.665,15.495,151.336
C08972=1104.292,297.289,-79.026,179.661,15.493,151.336
C08973=1104.288,297.040,-78.996,179.657,15.491,151.337
C08974=1104.282,296.792,-78.965,179.654,15.491,151.337
C08975=1104.276,296.544,-78.935,179.650,15.489,151.338
C08976=1104.270,296.296,-78.905,179.647,15.488,151.338
C08977=1104.265,296.048,-78.875,179.643,15.487,151.339
C08978=1104.259,295.800,-78.845,179.639,15.486,151.339
C08979=1104.253,295.552,-78.815,179.636,15.484,151.340
C08980=1104.248,295.304,-78.785,179.632,15.483,151.340
C08981=1104.242,295.056,-78.754,179.629,15.482,151.341
C08982=1104.236,294.807,-78.725,179.625,15.481,151.341
C08983=1104.230,294.560,-78.694,179.621,15.479,151.342
C08984=1104.225,294.311,-78.665,179.618,15.479,151.342
C08985=1104.219,294.063,-78.634,179.614,15.477,151.343
C08986=1104.214,293.815,-78.605,179.611,15.477,151.343
C08987=1104.208,293.567,-78.574,179.607,15.475,151.344
C08988=1104.202,293.319,-78.544,179.604,15.474,151.344
C08989=1104.196,293.071,-78.514,179.600,15.473,151.345
C08990=1104.191,292.823,-78.484,179.596,15.472,151.345
C08991=1104.185,292.575,-78.454,179.593,15.471,151.346
C08992=1104.180,292.326,-78.425,179.589,15.469,151.346
C08993=1104.174,292.078,-78.394,179.585,15.469,151.347
C08994=1104.168,291.830,-78.365,179.582,15.467,151.347
C08995=1104.162,291.582,-78.335,179.578,15.467,151.348
C08996=1104.157,291.334,-78.305,179.574,15.465,151.348
C08997=1104.151,291.086,-78.275,179.570,15.464,151.349
C08998=1104.146,290.837,-78.245,179.567,15.463,151.349
C08999=1104.139,290.589,-78.216,179.563,15.462,151.350
C09000=1104.134,290.342,-78.186,179.560,15.461,151.350
C09001=1104.126,289.976,-78.142,179.555,15.459,151.351
C09002=1104.118,289.610,-78.099,179.549,15.457,151.352
C09003=1104.109,289.244,-78.054,179.544,15.456,151.353
C09004=1104.101,288.878,-78.011,179.539,15.454,151.354
C09005=1104.096,288.630,-77.981,179.535,15.453,151.354
C09006=1104.089,288.382,-77.951,179.532,15.452,151.355
C09007=1104.083,288.134,-77.922,179.527,15.451,151.355
C09008=1104.078,287.885,-77.892,179.524,15.450,151.356
C09009=1104.072,287.637,-77.862,179.520,15.449,151.356
C09010=1104.066,287.389,-77.833,179.517,15.448,151.357
C09011=1104.061,287.142,-77.803,179.513,15.447,151.357
C09012=1104.055,286.893,-77.774,179.510,15.446,151.358
C09013=1104.049,286.645,-77.745,179.505,15.445,151.358
C09014=1104.044,286.397,-77.715,179.502,15.444,151.359
C09015=1104.038,286.148,-77.685,179.498,15.443,151.359
C09016=1104.033,285.900,-77.656,179.495,15.442,151.360
C09017=1104.026,285.652,-77.626,179.491,15.441,151.361
C09018=1104.021,285.405,-77.597,179.488,15.440,151.361
C09019=1104.016,285.156,-77.567,179.484,15.439,151.362
C09020=1104.009,284.908,-77.538,179.481,15.438,151.362
C09021=1104.004,284.660,-77.508,179.477,15.437,151.363
C09022=1103.998,284.411,-77.479,179.473,15.436,151.363
C09023=1103.993,284.164,-77.450,179.469,15.435,151.364
C09024=1103.987,283.915,-77.420,179.466,15.435,151.364
C09025=1103.982,283.667,-77.391,179.462,15.433,151.365
C09026=1103.975,283.419,-77.362,179.459,15.432,151.365
C09027=1103.970,283.170,-77.332,179.455,15.431,151.366
C09028=1103.964,282.923,-77.303,179.451,15.431,151.367
C09029=1103.959,282.674,-77.274,179.447,15.429,151.367
C09030=1103.954,282.425,-77.245,179.444,15.429,151.368
C09031=1103.947,282.177,-77.216,179.440,15.427,151.368
C09032=1103.942,281.929,-77.187,179.437,15.427,151.369
C09033=1103.937,281.681,-77.157,179.433,15.425,151.369
C09034=1103.931,281.433,-77.128,179.430,15.425,151.370
C09035=1103.925,281.184,-77.098,179.426,15.423,151.370
C09036=1103.920,280.937,-77.070,179.422,15.423,151.371
C09037=1103.914,280.688,-77.041,179.418,15.422,151.372
C09038=1103.908,280.440,-77.012,179.415,15.421,151.372
C09039=1103.903,280.191,-76.982,179.411,15.420,151.373
C09040=1103.897,279.944,-76.953,179.407,15.419,151.373
C09041=1103.891,279.696,-76.924,179.404,15.419,151.374
C09042=1103.885,279.447,-76.895,179.400,15.418,151.375
C09043=1103.880,279.199,-76.867,179.397,15.417,151.375
C09044=1103.874,278.951,-76.837,179.392,15.416,151.376
C09045=1103.868,278.703,-76.808,179.389,15.415,151.376
C09046=1103.863,278.454,-76.779,179.385,15.414,151.377
C09047=1103.857,278.206,-76.750,179.382,15.413,151.378
C09048=1103.851,277.958,-76.721,179.378,15.412,151.378
C09049=1103.846,277.709,-76.692,179.374,15.412,151.379
C09050=1103.840,277.462,-76.664,179.370,15.410,151.379
C09051=1103.835,277.213,-76.634,179.367,15.410,151.380
C09052=1103.829,276.964,-76.606,179.364,15.409,151.380
C09053=1103.821,276.609,-76.564,179.358,15.408,151.381
C09054=1103.812,276.252,-76.523,179.353,15.407,151.382
C09055=1103.804,275.896,-76.482,179.348,15.406,151.383
C09056=1103.797,275.539,-76.440,179.342,15.404,151.384
C09057=1103.791,275.291,-76.411,179.338,15.403,151.384
C09058=1103.785,275.042,-76.383,179.335,15.403,151.385
C09059=1103.779,274.795,-76.354,179.332,15.402,151.386
C09060=1103.774,274.546,-76.325,179.327,15.401,151.386
C09061=1103.768,274.298,-76.296,179.324,15.400,151.387
C09062=1103.762,274.050,-76.268,179.320,15.399,151.387
C09063=1103.757,273.801,-76.239,179.317,15.399,151.388
C09064=1103.751,273.553,-76.211,179.312,15.398,151.389
